			(*Robot 21*)
			IF (Human_Reqs_TraccTCP_R21)
					AND ((NOT Start_All_MTRobots AND NOT Start_All_BTRobots
					AND NOT Start_All_TCRobots AND NOT Start_All_TDRobots)
					OR (MAIN.R21.Task_ID_Ack=Tracc_TCP))
				THEN
					(*Start Robot*)
					Start_TraccTCP_21:= TRUE;
					(*Allow Robot to Proceed*)
					TraccRobot_21_Proceed:= TRUE;
			ELSE
					Start_TraccTCP_21:= FALSE;
					TraccRobot_21_Proceed:= FALSE;
			END_IF;	
			
			(*Robot 22*)
			IF (Human_Reqs_TraccTCP_R22)
					AND ((NOT Start_All_MTRobots AND NOT Start_All_BTRobots
					AND NOT Start_All_TCRobots AND NOT Start_All_TDRobots)
					OR (MAIN.R22.Task_ID_Ack=Tracc_TCP))
				THEN
					(*Start Robot*)
					Start_TraccTCP_22:= TRUE;
					(*Allow Robot to Proceed*)
					TraccRobot_22_Proceed:= TRUE;
			ELSE
					Start_TraccTCP_22:= FALSE;
					TraccRobot_22_Proceed:= FALSE;
			END_IF;	
			
			(*Robot 23*)
			IF (Human_Reqs_TraccTCP_R23)
					AND ((NOT Start_All_MTRobots AND NOT Start_All_BTRobots
					AND NOT Start_All_TCRobots AND NOT Start_All_TDRobots)
					OR (MAIN.R23.Task_ID_Ack=Tracc_TCP))
				THEN
					(*Start Robot*)
					Start_TraccTCP_23:= TRUE;
					(*Allow Robot to Proceed*)
					TraccRobot_23_Proceed:= TRUE;
			ELSE
					Start_TraccTCP_23:= FALSE;
					TraccRobot_23_Proceed:= FALSE;
			END_IF;	
			
			(*Robot 24*)
			IF (Human_Reqs_TraccTCP_R24)
					AND ((NOT Start_All_MTRobots AND NOT Start_All_BTRobots
					AND NOT Start_All_TCRobots AND NOT Start_All_TDRobots)
					OR (MAIN.R24.Task_ID_Ack=Tracc_TCP))
				THEN
					(*Start Robot*)
					Start_TraccTCP_24:= TRUE;
					(*Allow Robot to Proceed*)
					TraccRobot_24_Proceed:= TRUE;
			ELSE
					Start_TraccTCP_24:= FALSE;
					TraccRobot_24_Proceed:= FALSE;
			END_IF;	
			
			(*Robot 25*)
			IF (Human_Reqs_TraccTCP_R25)
					AND ((NOT Start_All_MTRobots AND NOT Start_All_BTRobots
					AND NOT Start_All_TCRobots AND NOT Start_All_TDRobots)
					OR (MAIN.R25.Task_ID_Ack=Tracc_TCP))
				THEN
					(*Start Robot*)
					Start_TraccTCP_25:= TRUE;
					(*Allow Robot to Proceed*)
					TraccRobot_25_Proceed:= TRUE;
			ELSE
					Start_TraccTCP_25:= FALSE;
					TraccRobot_25_Proceed:= FALSE;
			END_IF;	
			
			(*Robot 26*)
			IF (Human_Reqs_TraccTCP_R26)
					AND ((NOT Start_All_MTRobots AND NOT Start_All_BTRobots
					AND NOT Start_All_TCRobots AND NOT Start_All_TDRobots)
					OR (MAIN.R26.Task_ID_Ack=Tracc_TCP))
				THEN
					(*Start Robot*)
					Start_TraccTCP_26:= TRUE;
					(*Allow Robot to Proceed*)
					TraccRobot_26_Proceed:= TRUE;
			ELSE
					Start_TraccTCP_26:= FALSE;
					TraccRobot_26_Proceed:= FALSE;
			END_IF;	
			
			(*Robot 27*)
			IF (Human_Reqs_TraccTCP_R27)
					AND ((NOT Start_All_MTRobots AND NOT Start_All_BTRobots
					AND NOT Start_All_TCRobots AND NOT Start_All_TDRobots)
					OR (MAIN.R27.Task_ID_Ack=Tracc_TCP))
				THEN
					(*Start Robot*)
					Start_TraccTCP_27:= TRUE;
					(*Allow Robot to Proceed*)
					TraccRobot_27_Proceed:= TRUE;
			ELSE
					Start_TraccTCP_27:= FALSE;
					TraccRobot_27_Proceed:= FALSE;
			END_IF;	
			
			(*Robot 28*)
			IF (Human_Reqs_TraccTCP_R28)
					AND ((NOT Start_All_MTRobots AND NOT Start_All_BTRobots
					AND NOT Start_All_TCRobots AND NOT Start_All_TDRobots)
					OR (MAIN.R28.Task_ID_Ack=Tracc_TCP))
				THEN
					(*Start Robot*)
					Start_TraccTCP_28:= TRUE;
					(*Allow Robot to Proceed*)
					TraccRobot_28_Proceed:= TRUE;
			ELSE
					Start_TraccTCP_28:= FALSE;
					TraccRobot_28_Proceed:= FALSE;
			END_IF;	
			
			(*Robot 29*)
			IF (Human_Reqs_TraccTCP_R29)
					AND ((NOT Start_All_MTRobots AND NOT Start_All_BTRobots
					AND NOT Start_All_TCRobots AND NOT Start_All_TDRobots)
					OR (MAIN.R29.Task_ID_Ack=Tracc_TCP))
				THEN
					(*Start Robot*)
					Start_TraccTCP_29:= TRUE;
					(*Allow Robot to Proceed*)
					TraccRobot_29_Proceed:= TRUE;
			ELSE
					Start_TraccTCP_29:= FALSE;
					TraccRobot_29_Proceed:= FALSE;
			END_IF;
			
			(*Robot 30*)
			IF (Human_Reqs_TraccTCP_R30)
					AND ((NOT Start_All_MTRobots AND NOT Start_All_BTRobots
					AND NOT Start_All_TCRobots AND NOT Start_All_TDRobots)
					OR (MAIN.R30.Task_ID_Ack=Tracc_TCP))
				THEN
					(*Start Robot*)
					Start_TraccTCP_30:= TRUE;
					(*Allow Robot to Proceed*)
					TraccRobot_30_Proceed:= TRUE;
			ELSE
					Start_TraccTCP_30:= FALSE;
					TraccRobot_30_Proceed:= FALSE;
			END_IF;	
				

			
			
			
	ELSE
		Start_All_MTRobots:= FALSE;
		Start_All_BTRobots:= FALSE;
		Start_All_TCRobots:= FALSE;
		Start_All_TDRobots:= FALSE;
		Start_TDRobot_1:= FALSE;
		Start_TDRobot_2:= FALSE;
		Start_TDRobot_3:= FALSE;
		Start_TDRobot_4:= FALSE;
		Start_TDRobot_5:= FALSE;
		Start_TDRobot_6:= FALSE;
		Start_TDRobot_7:= FALSE;
		Start_TDRobot_8:= FALSE;
		Start_TDRobot_9:= FALSE;
		Start_TDRobot_10:= FALSE;
		Start_TDRobot_11:= FALSE;
		Start_TDRobot_12:= FALSE;
		Start_TDRobot_13:= FALSE;
		Start_TDRobot_14:= FALSE;
		Start_TDRobot_15:= FALSE;
		Start_TDRobot_16:= FALSE;
		Start_TDRobot_17:= FALSE;
		Start_TDRobot_18:= FALSE;
		Start_TDRobot_19:= FALSE;
		Start_TDRobot_20:= FALSE;
		Start_TDRobot_21:= FALSE;
		Start_TDRobot_22:= FALSE;
		Start_TDRobot_23:= FALSE;
		Start_TDRobot_24:= FALSE;
		Start_TDRobot_25:= FALSE;
		Start_TDRobot_26:= FALSE;
		Start_TDRobot_27:= FALSE;
		Start_TDRobot_28:= FALSE;
		Start_TDRobot_29:= FALSE;
		Start_TDRobot_30:= FALSE;
		Start_All_TraccTCP:= FALSE;
		Start_TraccTCP_1:= FALSE;
		Start_TraccTCP_2:= FALSE;
		Start_TraccTCP_3:= FALSE;
		Start_TraccTCP_4:= FALSE;
		Start_TraccTCP_5:= FALSE;
		Start_TraccTCP_6:= FALSE;
		Start_TraccTCP_7:= FALSE;
		Start_TraccTCP_8:= FALSE;
		Start_TraccTCP_9:= FALSE;
		Start_TraccTCP_10:= FALSE;
		Start_TraccTCP_11:= FALSE;
		Start_TraccTCP_12:= FALSE;
		Start_TraccTCP_13:= FALSE;
		Start_TraccTCP_14:= FALSE;
		Start_TraccTCP_15:= FALSE;
		Start_TraccTCP_16:= FALSE;
		Start_TraccTCP_17:= FALSE;
		Start_TraccTCP_18:= FALSE;
		Start_TraccTCP_19:= FALSE;
		Start_TraccTCP_20:= FALSE;
		Start_TraccTCP_21:= FALSE;
		Start_TraccTCP_22:= FALSE;
		Start_TraccTCP_23:= FALSE;
		Start_TraccTCP_24:= FALSE;
		Start_TraccTCP_25:= FALSE;
		Start_TraccTCP_26:= FALSE;
		Start_TraccTCP_27:= FALSE;
		Start_TraccTCP_28:= FALSE;
		Start_TraccTCP_29:= FALSE;
		Start_TraccTCP_30:= FALSE;
	END_IF;

(*---------------------------------------------------------------Completes----------------------------------------------------*)
	(*All Robots Complete Master Test*)
	IF Start_All_MTRobots AND All_Robots_Complete
		THEN
		Master_Tests_Complete:= TRUE;
		Human_Reqs_MasterTest:= FALSE;
		A_Robot_Reqs_MasterTest:= FALSE;
	END_IF;
	(*All Robots Complete Brake Test*)
	IF Start_All_BTRobots AND All_Robots_Complete
		THEN
		Brake_Tests_Complete:= TRUE;
		Human_Reqs_BrakeTest:= FALSE;
		A_Robot_Reqs_BrakeTest:= FALSE;
		All_RobotsReq_BrakeTest:= FALSE;
	END_IF;
	(*All Robots Complete Tip Change*)
	IF Start_All_TCRobots AND All_Robots_SteppersRST AND All_Robots_Complete
		THEN
		Tip_Change_Complete:= TRUE;
		Human_Reqs_TipChange:= FALSE;
	         Robot_Reqs_TipChange := FALSE;
	END_IF;

	(*All Robots Complete Tip Dress*)
	IF Start_All_TDRobots AND All_Robots_Complete
		THEN
		Tip_Dress_CompleteAll:= TRUE;
		TipChange_Reqs_TipDress:= FALSE;
		Robot_Reqs_TipDress:= FALSE;
	END_IF;

	(*Robot1 Complete Tip Dress*)
	IF Tip_Dress_Complete1
		THEN
		Human_Reqs_TipDressR1:= FALSE;
		Robot1_Reqs_TipDress:= FALSE;
	END_IF;

	(*Robot2 Complete Tip Dress*)
	IF Tip_Dress_Complete2
		THEN
		Human_Reqs_TipDressR2:= FALSE;
		Robot2_Reqs_TipDress:= FALSE;
	END_IF;

	(*Robot3 Complete Tip Dress*)
	IF Tip_Dress_Complete3
		THEN
		Human_Reqs_TipDressR3:= FALSE;
		Robot3_Reqs_TipDress:= FALSE;
	END_IF;

	(*Robot4 Complete Tip Dress*)
	IF Tip_Dress_Complete4
		THEN
		Human_Reqs_TipDressR4:= FALSE;
		Robot4_Reqs_TipDress:= FALSE;
	END_IF;

	(*Robot5 Complete Tip Dress*)
	IF Tip_Dress_Complete5
		THEN
		Human_Reqs_TipDressR5:= FALSE;
		Robot5_Reqs_TipDress:= FALSE;
	END_IF;

	(*Robot6 Complete Tip Dress*)
	IF Tip_Dress_Complete6
		THEN
		Human_Reqs_TipDressR6:= FALSE;
		Robot6_Reqs_TipDress:= FALSE;
	END_IF;

	(*Robot7 Complete Tip Dress*)
	IF Tip_Dress_Complete7
		THEN
		Human_Reqs_TipDressR7:= FALSE;
		Robot7_Reqs_TipDress:= FALSE;
	END_IF;

	(*Robot8 Complete Tip Dress*)
	IF Tip_Dress_Complete8
		THEN
		Human_Reqs_TipDressR8:= FALSE;
		Robot8_Reqs_TipDress:= FALSE;
	END_IF;

	(*Robot9 Complete Tip Dress*)
	IF Tip_Dress_Complete9
		THEN
		Human_Reqs_TipDressR9:= FALSE;
		Robot9_Reqs_TipDress:= FALSE;
	END_IF;

	(*Robot10 Complete Tip Dress*)
	IF Tip_Dress_Complete10
		THEN
		Human_Reqs_TipDressR10:= FALSE;
		Robot10_Reqs_TipDress:= FALSE;
	END_IF;

	(*Robot11 Complete Tip Dress*)
	IF Tip_Dress_Complete11
		THEN
		Human_Reqs_TipDressR11:= FALSE;
		Robot11_Reqs_TipDress:= FALSE;
	END_IF;

	(*Robot12 Complete Tip Dress*)
	IF Tip_Dress_Complete12
		THEN
		Human_Reqs_TipDressR12:= FALSE;
		Robot12_Reqs_TipDress:= FALSE;
	END_IF;

	(*Robot13 Complete Tip Dress*)
	IF Tip_Dress_Complete13
		THEN
		Human_Reqs_TipDressR13:= FALSE;
		Robot13_Reqs_TipDress:= FALSE;
	END_IF;

	(*Robot14 Complete Tip Dress*)
	IF Tip_Dress_Complete14
		THEN
		Human_Reqs_TipDressR14:= FALSE;
		Robot14_Reqs_TipDress:= FALSE;
	END_IF;

	(*Robot15 Complete Tip Dress*)
	IF Tip_Dress_Complete15
		THEN
		Human_Reqs_TipDressR15:= FALSE;
		Robot15_Reqs_TipDress:= FALSE;
	END_IF;

	(*Robot16 Complete Tip Dress*)
	IF Tip_Dress_Complete16
		THEN
		Human_Reqs_TipDressR16:= FALSE;
		Robot16_Reqs_TipDress:= FALSE;
	END_IF;

	(*Robot17 Complete Tip Dress*)
	IF Tip_Dress_Complete17
		THEN
		Human_Reqs_TipDressR17:= FALSE;
		Robot17_Reqs_TipDress:= FALSE;
	END_IF;

	(*Robot18 Complete Tip Dress*)
	IF Tip_Dress_Complete18
		THEN
		Human_Reqs_TipDressR18:= FALSE;
		Robot18_Reqs_TipDress:= FALSE;
	END_IF;

	(*Robot19 Complete Tip Dress*)
	IF Tip_Dress_Complete19
		THEN
		Human_Reqs_TipDressR19:= FALSE;
		Robot19_Reqs_TipDress:= FALSE;
	END_IF;

	(*Robot20 Complete Tip Dress*)
	IF Tip_Dress_Complete20
		THEN
		Human_Reqs_TipDressR20:= FALSE;
		Robot20_Reqs_TipDress:= FALSE;
	END_IF;

	(*Robot21 Complete Tip Dress*)
	IF Tip_Dress_Complete21
		THEN
		Human_Reqs_TipDressR21:= FALSE;
		Robot21_Reqs_TipDress:= FALSE;
	END_IF;

	(*Robot22 Complete Tip Dress*)
	IF Tip_Dress_Complete22
		THEN
		Human_Reqs_TipDressR22:= FALSE;
		Robot22_Reqs_TipDress:= FALSE;
	END_IF;

	(*Robot23 Complete Tip Dress*)
	IF Tip_Dress_Complete23
		THEN
		Human_Reqs_TipDressR23:= FALSE;
		Robot23_Reqs_TipDress:= FALSE;
	END_IF;

	(*Robot24 Complete Tip Dress*)
	IF Tip_Dress_Complete24
		THEN
		Human_Reqs_TipDressR24:= FALSE;
		Robot24_Reqs_TipDress:= FALSE;
	END_IF;

	(*Robot25 Complete Tip Dress*)
	IF Tip_Dress_Complete25
		THEN
		Human_Reqs_TipDressR25:= FALSE;
		Robot25_Reqs_TipDress:= FALSE;
	END_IF;

	(*Robot26 Complete Tip Dress*)
	IF Tip_Dress_Complete26
		THEN
		Human_Reqs_TipDressR26:= FALSE;
		Robot26_Reqs_TipDress:= FALSE;
	END_IF;

	(*Robot27 Complete Tip Dress*)
	IF Tip_Dress_Complete27
		THEN
		Human_Reqs_TipDressR27:= FALSE;
		Robot27_Reqs_TipDress:= FALSE;
	END_IF;

	(*Robot28 Complete Tip Dress*)
	IF Tip_Dress_Complete28
		THEN
		Human_Reqs_TipDressR28:= FALSE;
		Robot28_Reqs_TipDress:= FALSE;
	END_IF;

	(*Robot29 Complete Tip Dress*)
	IF Tip_Dress_Complete29
		THEN
		Human_Reqs_TipDressR29:= FALSE;
		Robot29_Reqs_TipDress:= FALSE;
	END_IF;

	(*Robot30 Complete Tip Dress*)
	IF Tip_Dress_Complete30
		THEN
		Human_Reqs_TipDressR30:= FALSE;
		Robot30_Reqs_TipDress:= FALSE;
	END_IF;

	(*Robot 1 Complete TraccTCP*)
	IF TraccTCP_Complete1
		THEN
		Human_Reqs_TraccTCP_R1:= FALSE;
		Robot1_Reqs_TraccTCP:= FALSE;
	END_IF;

	(*Robot 2 Complete TraccTCP*)
	IF TraccTCP_Complete2
		THEN
		Human_Reqs_TraccTCP_R2:= FALSE;
		Robot2_Reqs_TraccTCP:= FALSE;
	END_IF;

	(*Robot 3 Complete TraccTCP*)
	IF TraccTCP_Complete3
		THEN
		Human_Reqs_TraccTCP_R3:= FALSE;
		Robot3_Reqs_TraccTCP:= FALSE;
	END_IF;

	(*Robot 4 Complete TraccTCP*)
	IF TraccTCP_Complete4
		THEN
		Human_Reqs_TraccTCP_R4:= FALSE;
		Robot4_Reqs_TraccTCP:= FALSE;
	END_IF;	

	(*Robot 5 Complete TraccTCP*)
	IF TraccTCP_Complete5
		THEN
		Human_Reqs_TraccTCP_R5:= FALSE;
		Robot5_Reqs_TraccTCP:= FALSE;
	END_IF;

	(*Robot 6 Complete TraccTCP*)
	IF TraccTCP_Complete6
		THEN
		Human_Reqs_TraccTCP_R6:= FALSE;
		Robot6_Reqs_TraccTCP:= FALSE;
	END_IF;

	(*Robot 7 Complete TraccTCP*)
	IF TraccTCP_Complete7
		THEN
		Human_Reqs_TraccTCP_R7:= FALSE;
		Robot7_Reqs_TraccTCP:= FALSE;
	END_IF;
	
	(*Robot 8 Complete TraccTCP*)
	IF TraccTCP_Complete8
		THEN
		Human_Reqs_TraccTCP_R8:= FALSE;
		Robot8_Reqs_TraccTCP:= FALSE;
	END_IF;
	
	(*Robot 9 Complete TraccTCP*)
	IF TraccTCP_Complete9
		THEN
		Human_Reqs_TraccTCP_R9:= FALSE;
		Robot9_Reqs_TraccTCP:= FALSE;
	END_IF;
	
	(*Robot 10 Complete TraccTCP*)
	IF TraccTCP_Complete10
		THEN
		Human_Reqs_TraccTCP_R10:= FALSE;
		Robot10_Reqs_TraccTCP:= FALSE;
	END_IF;

	(*Robot 11 Complete TraccTCP*)
	IF TraccTCP_Complete11
		THEN
		Human_Reqs_TraccTCP_R11:= FALSE;
		Robot11_Reqs_TraccTCP:= FALSE;
	END_IF;
	
	(*Robot 12 Complete TraccTCP*)
	IF TraccTCP_Complete12
		THEN
		Human_Reqs_TraccTCP_R12:= FALSE;
		Robot12_Reqs_TraccTCP:= FALSE;
	END_IF;
	
	(*Robot 13 Complete TraccTCP*)
	IF TraccTCP_Complete13
		THEN
		Human_Reqs_TraccTCP_R13:= FALSE;
		Robot13_Reqs_TraccTCP:= FALSE;
	END_IF;
	
	(*Robot 14 Complete TraccTCP*)
	IF TraccTCP_Complete14
		THEN
		Human_Reqs_TraccTCP_R14:= FALSE;
		Robot14_Reqs_TraccTCP:= FALSE;
	END_IF;
	
	(*Robot 15 Complete TraccTCP*)
	IF TraccTCP_Complete15
		THEN
		Human_Reqs_TraccTCP_R15:= FALSE;
		Robot15_Reqs_TraccTCP:= FALSE;
	END_IF;
	
	(*Robot 16 Complete TraccTCP*)
	IF TraccTCP_Complete16
		THEN
		Human_Reqs_TraccTCP_R16:= FALSE;
		Robot16_Reqs_TraccTCP:= FALSE;
	END_IF;
	
	(*Robot 17 Complete TraccTCP*)
	IF TraccTCP_Complete17
		THEN
		Human_Reqs_TraccTCP_R17:= FALSE;
		Robot17_Reqs_TraccTCP:= FALSE;
	END_IF;
	
	(*Robot 18 Complete TraccTCP*)
	IF TraccTCP_Complete18
		THEN
		Human_Reqs_TraccTCP_R18:= FALSE;
		Robot18_Reqs_TraccTCP:= FALSE;
	END_IF;
	
	(*Robot 19 Complete TraccTCP*)
	IF TraccTCP_Complete19
		THEN
		Human_Reqs_TraccTCP_R19:= FALSE;
		Robot19_Reqs_TraccTCP:= FALSE;
	END_IF;
	
	(*Robot 20 Complete TraccTCP*)
	IF TraccTCP_Complete20
		THEN
		Human_Reqs_TraccTCP_R20:= FALSE;
		Robot20_Reqs_TraccTCP:= FALSE;
	END_IF;

	(*Robot 21 Complete TraccTCP*)
	IF TraccTCP_Complete21
		THEN
		Human_Reqs_TraccTCP_R21:= FALSE;
		Robot21_Reqs_TraccTCP:= FALSE;
	END_IF;
	
	(*Robot 22 Complete TraccTCP*)
	IF TraccTCP_Complete22
		THEN
		Human_Reqs_TraccTCP_R22:= FALSE;
		Robot22_Reqs_TraccTCP:= FALSE;
	END_IF;
	
	(*Robot 23 Complete TraccTCP*)
	IF TraccTCP_Complete23
		THEN
		Human_Reqs_TraccTCP_R23:= FALSE;
		Robot23_Reqs_TraccTCP:= FALSE;
	END_IF;
	
	(*Robot 24 Complete TraccTCP*)
	IF TraccTCP_Complete24
		THEN
		Human_Reqs_TraccTCP_R24:= FALSE;
		Robot24_Reqs_TraccTCP:= FALSE;
	END_IF;
	
	(*Robot 25 Complete TraccTCP*)
	IF TraccTCP_Complete25
		THEN
		Human_Reqs_TraccTCP_R25:= FALSE;
		Robot25_Reqs_TraccTCP:= FALSE;
	END_IF;
	
	(*Robot 26 Complete TraccTCP*)
	IF TraccTCP_Complete26
		THEN
		Human_Reqs_TraccTCP_R26:= FALSE;
		Robot26_Reqs_TraccTCP:= FALSE;
	END_IF;
	
	(*Robot 27 Complete TraccTCP*)
	IF TraccTCP_Complete27
		THEN
		Human_Reqs_TraccTCP_R27:= FALSE;
		Robot27_Reqs_TraccTCP:= FALSE;
	END_IF;
	
	(*Robot 28 Complete TraccTCP*)
	IF TraccTCP_Complete28
		THEN
		Human_Reqs_TraccTCP_R28:= FALSE;
		Robot28_Reqs_TraccTCP:= FALSE;
	END_IF;
	
	(*Robot 29 Complete TraccTCP*)
	IF TraccTCP_Complete29
		THEN
		Human_Reqs_TraccTCP_R29:= FALSE;
		Robot29_Reqs_TraccTCP:= FALSE;
	END_IF;
	
	(*Robot 30 Complete TraccTCP*)
	IF TraccTCP_Complete30
		THEN
		Human_Reqs_TraccTCP_R30:= FALSE;
		Robot30_Reqs_TraccTCP:= FALSE;
	END_IF;
	
	
	
(*!!!!!!!!!!!!!!!!!!!!!!!!!!!!!!!!!!!!!!!!!!!!!!!!!!!!!!!!!!!!!!!!!!!!!!!!!!!!!!!!!!!!!!!!!!!!!!!!! Cycle Complete !!!!!!!!!!!!!!!!!!!!!!!!!!!!!!!!!!!!!!!!!!!!!!!!!!!!!!!!!!!!!!!!!!!!!!!!!!!!!!!!!!!!!!!!!!*)
	(*Set Cycle Complete*)
	IF Auto_Run AND (Master_Tests_Complete OR Brake_Tests_Complete OR Tip_Change_Complete OR Tip_Dress_CompleteAll OR TraccTCP_CompleteAll)
		THEN Cycle_Complete:= TRUE;
	END_IF;
	(*Reset All Completes*)
	IF Cycle_Complete AND All_Robots_Clear
		THEN
					Reset_All_Completes:= TRUE;
	END_IF;
	(*Perform Actual Reset*)
		IF Reset_All_Completes
			THEN
				Cycle_Complete:= FALSE;
				Human_Reqs_MasterTest := FALSE;
				A_Robot_Reqs_MasterTest :=FALSE;
				Master_Tests_Complete:= FALSE;
				Human_Reqs_BrakeTest := FALSE;
				A_Robot_Reqs_BrakeTest := FALSE;
				All_RobotsReq_BrakeTest := FALSE;
				Brake_Tests_Complete:= FALSE;
				Tip_Change_Complete:= FALSE;
				Tip_Dress_CompleteAll:= FALSE;
				TraccTCP_CompleteAll:= FALSE;
				Reset_All_Completes:= FALSE;
		END_IF;

(*$$$$$$$$$$$$$$$$$$$$$$$$$$$$$$$$$$$ Production Counter $$$$$$$$$$$$$$$$$$$$$$$$$$$$$$$$$$$$$$$$$$*)
	(*Increment Tip Change Counter*)
	Prod_Inc.CLK:= Tip_Change_Complete;
	Prod_Inc();
	IF Prod_Inc.Q
		THEN
		Production_Count:= Production_Count+1;
	END_IF;
	IF Discrete_In.ResetProd
		THEN
		Production_Count:= 0;
	END_IF;
	Prod_Count_Out:= Production_Count;
(*~~~~~~~~~~~~~~~~~~~~~~~~~~~~~~~~ Cycle Time Counters ~~~~~~~~~~~~~~~~~~~~~~~~~*)
	(*Move Previous To Register*)
	Cycle_Time_Pulse.CLK:= Tip_Change_Complete;
	Cycle_Time_Pulse();
	IF Cycle_Time_Pulse.Q
		THEN
		PrevCycle_Time_Out:= Cycle_Time_Out;
	END_IF;
	(*Monitor Current Cycle Time*)
		Cycle_Time.PT:= T#9999S;
		Cycle_Time.IN:= Auto_Run AND NOT Cycle_Complete;
		Cycle_Time();
		Cycle_Time_Out:= Cycle_Time.ET;

(*^^^^^^^^^^^^^^^^^^^^^^^^^^^^^^^^^^^^^^ General Visualization ^^^^^^^^^^^^^^^^^^^^^^^^^^^^^^^^^^^^*)

(*#################################### Register Robots to Tool ##################################*)
(*+++++++++++THIS AREA IS CUSTOM PER INSTALLATION AND WILL HAVE TO BE MODIFIED PER +++++++++++++*)
(*+++++++++++THIS AREA IS CUSTOM PER INSTALLATION AND WILL HAVE TO BE MODIFIED PER +++++++++++++*)

	(*Data From All Robot(s)*)

	All_Robots_Clear:= MAIN.R1.Clear_Of_EquipInterf8 AND MAIN.R1.Task_ID_Ack<350 AND
					(MAIN.R2.Clear_Of_EquipInterf8 AND MAIN.R2.Task_ID_Ack<350 OR GTAC_CONFIG.Option_Robot_Count<2) AND
					(MAIN.R3.Clear_Of_EquipInterf8 AND MAIN.R3.Task_ID_Ack<350 OR GTAC_CONFIG.Option_Robot_Count<3) AND
					(MAIN.R4.Clear_Of_EquipInterf8 AND MAIN.R4.Task_ID_Ack<350 OR GTAC_CONFIG.Option_Robot_Count<4) AND
					(MAIN.R5.Clear_Of_EquipInterf8 AND MAIN.R5.Task_ID_Ack<350 OR GTAC_CONFIG.Option_Robot_Count<5) AND
					(MAIN.R6.Clear_Of_EquipInterf8 AND MAIN.R6.Task_ID_Ack<350 OR GTAC_CONFIG.Option_Robot_Count<6) AND
					(MAIN.R7.Clear_Of_EquipInterf8 AND MAIN.R7.Task_ID_Ack<350 OR GTAC_CONFIG.Option_Robot_Count<7) AND
					(MAIN.R8.Clear_Of_EquipInterf8 AND MAIN.R8.Task_ID_Ack<350 OR GTAC_CONFIG.Option_Robot_Count<8) AND
					(MAIN.R9.Clear_Of_EquipInterf8 AND MAIN.R9.Task_ID_Ack<350 OR GTAC_CONFIG.Option_Robot_Count<9) AND
					(MAIN.R10.Clear_Of_EquipInterf8 AND MAIN.R10.Task_ID_Ack<350 OR GTAC_CONFIG.Option_Robot_Count<10) AND
					(MAIN.R11.Clear_Of_EquipInterf8 AND MAIN.R11.Task_ID_Ack<350 OR GTAC_CONFIG.Option_Robot_Count<11) AND
					(MAIN.R12.Clear_Of_EquipInterf8 AND MAIN.R12.Task_ID_Ack<350 OR GTAC_CONFIG.Option_Robot_Count<12) AND
					(MAIN.R13.Clear_Of_EquipInterf8 AND MAIN.R13.Task_ID_Ack<350 OR GTAC_CONFIG.Option_Robot_Count<13) AND
					(MAIN.R14.Clear_Of_EquipInterf8 AND MAIN.R14.Task_ID_Ack<350 OR GTAC_CONFIG.Option_Robot_Count<14) AND
					(MAIN.R15.Clear_Of_EquipInterf8 AND MAIN.R15.Task_ID_Ack<350 OR GTAC_CONFIG.Option_Robot_Count<15) AND
					(MAIN.R16.Clear_Of_EquipInterf8 AND MAIN.R16.Task_ID_Ack<350 OR GTAC_CONFIG.Option_Robot_Count<16) AND
					(MAIN.R17.Clear_Of_EquipInterf8 AND MAIN.R17.Task_ID_Ack<350 OR GTAC_CONFIG.Option_Robot_Count<17) AND
					(MAIN.R18.Clear_Of_EquipInterf8 AND MAIN.R18.Task_ID_Ack<350 OR GTAC_CONFIG.Option_Robot_Count<18) AND
					(MAIN.R19.Clear_Of_EquipInterf8 AND MAIN.R19.Task_ID_Ack<350 OR GTAC_CONFIG.Option_Robot_Count<19) AND
					(MAIN.R20.Clear_Of_EquipInterf8 AND MAIN.R20.Task_ID_Ack<350 OR GTAC_CONFIG.Option_Robot_Count<20) AND
					(MAIN.R21.Clear_Of_EquipInterf8 AND MAIN.R21.Task_ID_Ack<350 OR GTAC_CONFIG.Option_Robot_Count<21) AND
					(MAIN.R22.Clear_Of_EquipInterf8 AND MAIN.R22.Task_ID_Ack<350 OR GTAC_CONFIG.Option_Robot_Count<22) AND
					(MAIN.R23.Clear_Of_EquipInterf8 AND MAIN.R23.Task_ID_Ack<350 OR GTAC_CONFIG.Option_Robot_Count<23) AND
					(MAIN.R24.Clear_Of_EquipInterf8 AND MAIN.R24.Task_ID_Ack<350 OR GTAC_CONFIG.Option_Robot_Count<24) AND
					(MAIN.R25.Clear_Of_EquipInterf8 AND MAIN.R25.Task_ID_Ack<350 OR GTAC_CONFIG.Option_Robot_Count<25) AND
					(MAIN.R26.Clear_Of_EquipInterf8 AND MAIN.R26.Task_ID_Ack<350 OR GTAC_CONFIG.Option_Robot_Count<26) AND
					(MAIN.R27.Clear_Of_EquipInterf8 AND MAIN.R27.Task_ID_Ack<350 OR GTAC_CONFIG.Option_Robot_Count<27) AND
					(MAIN.R28.Clear_Of_EquipInterf8 AND MAIN.R28.Task_ID_Ack<350 OR GTAC_CONFIG.Option_Robot_Count<28) AND
					(MAIN.R29.Clear_Of_EquipInterf8 AND MAIN.R29.Task_ID_Ack<350 OR GTAC_CONFIG.Option_Robot_Count<29) AND
					(MAIN.R30.Clear_Of_EquipInterf8 AND MAIN.R30.Task_ID_Ack<350 OR GTAC_CONFIG.Option_Robot_Count<30);

	All_Robots_WorkingOK:=  (Start_All_MTRobots AND MAIN.R1.Task_ID_Ack=Master_Test AND MAIN.R1.Operating AND
											(MAIN.R2.Task_ID_Ack=Master_Test AND MAIN.R2.Operating OR GTAC_CONFIG.Option_Robot_Count<2) AND
											(MAIN.R3.Task_ID_Ack=Master_Test AND MAIN.R3.Operating OR GTAC_CONFIG.Option_Robot_Count<3) AND
											(MAIN.R4.Task_ID_Ack=Master_Test AND MAIN.R4.Operating OR GTAC_CONFIG.Option_Robot_Count<4) AND
											(MAIN.R5.Task_ID_Ack=Master_Test AND MAIN.R5.Operating OR GTAC_CONFIG.Option_Robot_Count<5) AND
											(MAIN.R6.Task_ID_Ack=Master_Test AND MAIN.R6.Operating OR GTAC_CONFIG.Option_Robot_Count<6) AND
											(MAIN.R7.Task_ID_Ack=Master_Test AND MAIN.R7.Operating OR GTAC_CONFIG.Option_Robot_Count<7) AND
											(MAIN.R8.Task_ID_Ack= Master_Test AND MAIN.R8.Operating OR GTAC_CONFIG.Option_Robot_Count<8) AND
											(MAIN.R9.Task_ID_Ack=Master_Test AND MAIN.R9.Operating OR GTAC_CONFIG.Option_Robot_Count<9) AND
											(MAIN.R10.Task_ID_Ack= Master_Test AND MAIN.R10.Operating OR GTAC_CONFIG.Option_Robot_Count<10) AND
											(MAIN.R11.Task_ID_Ack=Master_Test AND MAIN.R11.Operating OR GTAC_CONFIG.Option_Robot_Count<11) AND
											(MAIN.R12.Task_ID_Ack=Master_Test AND MAIN.R12.Operating OR GTAC_CONFIG.Option_Robot_Count<12) AND
											(MAIN.R13.Task_ID_Ack=Master_Test AND MAIN.R13.Operating OR GTAC_CONFIG.Option_Robot_Count<13) AND
											(MAIN.R14.Task_ID_Ack=Master_Test AND MAIN.R14.Operating OR GTAC_CONFIG.Option_Robot_Count<14) AND
											(MAIN.R15.Task_ID_Ack=Master_Test AND MAIN.R15.Operating OR GTAC_CONFIG.Option_Robot_Count<15) AND
											(MAIN.R16.Task_ID_Ack=Master_Test AND MAIN.R16.Operating OR GTAC_CONFIG.Option_Robot_Count<16) AND
											(MAIN.R17.Task_ID_Ack=Master_Test AND MAIN.R17.Operating OR GTAC_CONFIG.Option_Robot_Count<17) AND
											(MAIN.R18.Task_ID_Ack= Master_Test AND MAIN.R18.Operating OR GTAC_CONFIG.Option_Robot_Count<18) AND
											(MAIN.R19.Task_ID_Ack=Master_Test AND MAIN.R19.Operating OR GTAC_CONFIG.Option_Robot_Count<19) AND
											(MAIN.R20.Task_ID_Ack=Master_Test AND MAIN.R20.Operating OR GTAC_CONFIG.Option_Robot_Count<20) AND
											(MAIN.R21.Task_ID_Ack=Master_Test AND MAIN.R21.Operating OR GTAC_CONFIG.Option_Robot_Count<21) AND
											(MAIN.R22.Task_ID_Ack=Master_Test AND MAIN.R22.Operating OR GTAC_CONFIG.Option_Robot_Count<22) AND
											(MAIN.R23.Task_ID_Ack=Master_Test AND MAIN.R23.Operating OR GTAC_CONFIG.Option_Robot_Count<23) AND
											(MAIN.R24.Task_ID_Ack=Master_Test AND MAIN.R24.Operating OR GTAC_CONFIG.Option_Robot_Count<24) AND
											(MAIN.R25.Task_ID_Ack=Master_Test AND MAIN.R25.Operating OR GTAC_CONFIG.Option_Robot_Count<25) AND
											(MAIN.R26.Task_ID_Ack=Master_Test AND MAIN.R26.Operating OR GTAC_CONFIG.Option_Robot_Count<26) AND
											(MAIN.R27.Task_ID_Ack=Master_Test AND MAIN.R27.Operating OR GTAC_CONFIG.Option_Robot_Count<27) AND
											(MAIN.R28.Task_ID_Ack=Master_Test AND MAIN.R28.Operating OR GTAC_CONFIG.Option_Robot_Count<28) AND
											(MAIN.R29.Task_ID_Ack=Master_Test AND MAIN.R29.Operating OR GTAC_CONFIG.Option_Robot_Count<29) AND
											(MAIN.R30.Task_ID_Ack=Master_Test AND MAIN.R30.Operating OR GTAC_CONFIG.Option_Robot_Count<30))
											OR
							(Start_All_BTRobots AND MAIN.R1.Task_ID_Ack=Brake_Test AND MAIN.R1.Operating AND
											(MAIN.R2.Task_ID_Ack=Brake_Test AND MAIN.R2.Operating OR GTAC_CONFIG.Option_Robot_Count<2) AND
											(MAIN.R3.Task_ID_Ack=Brake_Test AND MAIN.R3.Operating OR GTAC_CONFIG.Option_Robot_Count<3) AND
											(MAIN.R4.Task_ID_Ack=Brake_Test AND MAIN.R4.Operating OR GTAC_CONFIG.Option_Robot_Count<4) AND
											(MAIN.R5.Task_ID_Ack=Brake_Test AND MAIN.R5.Operating OR GTAC_CONFIG.Option_Robot_Count<5) AND
											(MAIN.R6.Task_ID_Ack=Brake_Test AND MAIN.R6.Operating OR GTAC_CONFIG.Option_Robot_Count<6) AND
											(MAIN.R7.Task_ID_Ack=Brake_Test AND MAIN.R7.Operating OR GTAC_CONFIG.Option_Robot_Count<7) AND
											(MAIN.R8.Task_ID_Ack=Brake_Test AND MAIN.R8.Operating OR GTAC_CONFIG.Option_Robot_Count<8) AND
											(MAIN.R9.Task_ID_Ack=Brake_Test AND MAIN.R9.Operating OR GTAC_CONFIG.Option_Robot_Count<9) AND
											(MAIN.R10.Task_ID_Ack=Brake_Test AND MAIN.R10.Operating OR GTAC_CONFIG.Option_Robot_Count<10) AND
											(MAIN.R11.Task_ID_Ack=Brake_Test AND MAIN.R11.Operating OR GTAC_CONFIG.Option_Robot_Count<11) AND
											(MAIN.R12.Task_ID_Ack=Brake_Test AND MAIN.R12.Operating OR GTAC_CONFIG.Option_Robot_Count<12) AND
											(MAIN.R13.Task_ID_Ack=Brake_Test AND MAIN.R13.Operating OR GTAC_CONFIG.Option_Robot_Count<13) AND
											(MAIN.R14.Task_ID_Ack=Brake_Test AND MAIN.R14.Operating OR GTAC_CONFIG.Option_Robot_Count<14) AND
											(MAIN.R15.Task_ID_Ack=Brake_Test AND MAIN.R15.Operating OR GTAC_CONFIG.Option_Robot_Count<15) AND
											(MAIN.R16.Task_ID_Ack=Brake_Test AND MAIN.R16.Operating OR GTAC_CONFIG.Option_Robot_Count<16) AND
											(MAIN.R17.Task_ID_Ack=Brake_Test AND MAIN.R17.Operating OR GTAC_CONFIG.Option_Robot_Count<17) AND
											(MAIN.R18.Task_ID_Ack=Brake_Test AND MAIN.R18.Operating OR GTAC_CONFIG.Option_Robot_Count<18) AND
											(MAIN.R19.Task_ID_Ack=Brake_Test AND MAIN.R19.Operating OR GTAC_CONFIG.Option_Robot_Count<19) AND
											(MAIN.R20.Task_ID_Ack=Brake_Test AND MAIN.R20.Operating OR GTAC_CONFIG.Option_Robot_Count<20) AND
											(MAIN.R21.Task_ID_Ack=Brake_Test AND MAIN.R21.Operating OR GTAC_CONFIG.Option_Robot_Count<21) AND
											(MAIN.R22.Task_ID_Ack=Brake_Test AND MAIN.R22.Operating OR GTAC_CONFIG.Option_Robot_Count<22) AND
											(MAIN.R23.Task_ID_Ack=Brake_Test AND MAIN.R23.Operating OR GTAC_CONFIG.Option_Robot_Count<23) AND
											(MAIN.R24.Task_ID_Ack=Brake_Test AND MAIN.R24.Operating OR GTAC_CONFIG.Option_Robot_Count<24) AND
											(MAIN.R25.Task_ID_Ack=Brake_Test AND MAIN.R25.Operating OR GTAC_CONFIG.Option_Robot_Count<25) AND
											(MAIN.R26.Task_ID_Ack=Brake_Test AND MAIN.R26.Operating OR GTAC_CONFIG.Option_Robot_Count<26) AND
											(MAIN.R27.Task_ID_Ack=Brake_Test AND MAIN.R27.Operating OR GTAC_CONFIG.Option_Robot_Count<27) AND
											(MAIN.R28.Task_ID_Ack=Brake_Test AND MAIN.R28.Operating OR GTAC_CONFIG.Option_Robot_Count<28) AND
											(MAIN.R29.Task_ID_Ack=Brake_Test AND MAIN.R29.Operating OR GTAC_CONFIG.Option_Robot_Count<29) AND
											(MAIN.R30.Task_ID_Ack=Brake_Test AND MAIN.R30.Operating OR GTAC_CONFIG.Option_Robot_Count<30))
											OR
							(Start_All_TCRobots AND MAIN.R1.Task_ID_Ack=Tip_Change AND MAIN.R1.Operating AND
											(MAIN.R2.Task_ID_Ack=Tip_Change AND MAIN.R2.Operating OR GTAC_CONFIG.Option_Robot_Count<2) AND
											(MAIN.R3.Task_ID_Ack=Tip_Change AND MAIN.R3.Operating OR GTAC_CONFIG.Option_Robot_Count<3) AND
											(MAIN.R4.Task_ID_Ack=Tip_Change AND MAIN.R4.Operating OR GTAC_CONFIG.Option_Robot_Count<4) AND
											(MAIN.R5.Task_ID_Ack=Tip_Change AND MAIN.R5.Operating OR GTAC_CONFIG.Option_Robot_Count<5) AND
											(MAIN.R6.Task_ID_Ack=Tip_Change AND MAIN.R6.Operating OR GTAC_CONFIG.Option_Robot_Count<6) AND
											(MAIN.R7.Task_ID_Ack=Tip_Change AND MAIN.R7.Operating OR GTAC_CONFIG.Option_Robot_Count<7) AND
											(MAIN.R8.Task_ID_Ack=Tip_Change AND MAIN.R8.Operating OR GTAC_CONFIG.Option_Robot_Count<8) AND
											(MAIN.R9.Task_ID_Ack=Tip_Change AND MAIN.R9.Operating OR GTAC_CONFIG.Option_Robot_Count<9) AND
											(MAIN.R10.Task_ID_Ack=Tip_Change AND MAIN.R10.Operating OR GTAC_CONFIG.Option_Robot_Count<10) AND
											(MAIN.R11.Task_ID_Ack=Tip_Change AND MAIN.R11.Operating OR GTAC_CONFIG.Option_Robot_Count<11) AND
											(MAIN.R12.Task_ID_Ack=Tip_Change AND MAIN.R12.Operating OR GTAC_CONFIG.Option_Robot_Count<12) AND
											(MAIN.R13.Task_ID_Ack=Tip_Change AND MAIN.R13.Operating OR GTAC_CONFIG.Option_Robot_Count<13) AND
											(MAIN.R14.Task_ID_Ack=Tip_Change AND MAIN.R14.Operating OR GTAC_CONFIG.Option_Robot_Count<14) AND
											(MAIN.R15.Task_ID_Ack=Tip_Change AND MAIN.R15.Operating OR GTAC_CONFIG.Option_Robot_Count<15) AND
											(MAIN.R16.Task_ID_Ack=Tip_Change AND MAIN.R16.Operating OR GTAC_CONFIG.Option_Robot_Count<16) AND
											(MAIN.R17.Task_ID_Ack=Tip_Change AND MAIN.R17.Operating OR GTAC_CONFIG.Option_Robot_Count<17) AND
											(MAIN.R18.Task_ID_Ack=Tip_Change AND MAIN.R18.Operating OR GTAC_CONFIG.Option_Robot_Count<18) AND
											(MAIN.R19.Task_ID_Ack=Tip_Change AND MAIN.R19.Operating OR GTAC_CONFIG.Option_Robot_Count<19) AND
											(MAIN.R20.Task_ID_Ack=Tip_Change AND MAIN.R20.Operating OR GTAC_CONFIG.Option_Robot_Count<20) AND
											(MAIN.R21.Task_ID_Ack=Tip_Change AND MAIN.R21.Operating OR GTAC_CONFIG.Option_Robot_Count<21) AND
											(MAIN.R22.Task_ID_Ack=Tip_Change AND MAIN.R22.Operating OR GTAC_CONFIG.Option_Robot_Count<22) AND
											(MAIN.R23.Task_ID_Ack=Tip_Change AND MAIN.R23.Operating OR GTAC_CONFIG.Option_Robot_Count<23) AND
											(MAIN.R24.Task_ID_Ack=Tip_Change AND MAIN.R24.Operating OR GTAC_CONFIG.Option_Robot_Count<24) AND
											(MAIN.R25.Task_ID_Ack=Tip_Change AND MAIN.R25.Operating OR GTAC_CONFIG.Option_Robot_Count<25) AND
											(MAIN.R26.Task_ID_Ack=Tip_Change AND MAIN.R26.Operating OR GTAC_CONFIG.Option_Robot_Count<26) AND
											(MAIN.R27.Task_ID_Ack=Tip_Change AND MAIN.R27.Operating OR GTAC_CONFIG.Option_Robot_Count<27) AND
											(MAIN.R28.Task_ID_Ack=Tip_Change AND MAIN.R28.Operating OR GTAC_CONFIG.Option_Robot_Count<28) AND
											(MAIN.R29.Task_ID_Ack=Tip_Change AND MAIN.R29.Operating OR GTAC_CONFIG.Option_Robot_Count<29) AND
											(MAIN.R30.Task_ID_Ack=Tip_Change AND MAIN.R30.Operating OR GTAC_CONFIG.Option_Robot_Count<30))
											OR
							(Start_All_TDRobots AND MAIN.R1.Task_ID_Ack=Tip_Dress AND MAIN.R1.Operating AND
											(MAIN.R2.Task_ID_Ack=Tip_Dress AND MAIN.R2.Operating OR GTAC_CONFIG.Option_Robot_Count<2) AND
											(MAIN.R3.Task_ID_Ack=Tip_Dress AND MAIN.R3.Operating OR GTAC_CONFIG.Option_Robot_Count<3) AND
											(MAIN.R4.Task_ID_Ack=Tip_Dress AND MAIN.R4.Operating OR GTAC_CONFIG.Option_Robot_Count<4) AND
											(MAIN.R5.Task_ID_Ack=Tip_Dress AND MAIN.R5.Operating OR GTAC_CONFIG.Option_Robot_Count<5) AND
											(MAIN.R6.Task_ID_Ack=Tip_Dress AND MAIN.R6.Operating OR GTAC_CONFIG.Option_Robot_Count<6) AND
											(MAIN.R7.Task_ID_Ack=Tip_Dress AND MAIN.R7.Operating OR GTAC_CONFIG.Option_Robot_Count<7) AND
											(MAIN.R8.Task_ID_Ack=Tip_Dress AND MAIN.R8.Operating OR GTAC_CONFIG.Option_Robot_Count<8) AND
											(MAIN.R9.Task_ID_Ack=Tip_Dress AND MAIN.R9.Operating OR GTAC_CONFIG.Option_Robot_Count<9) AND
											(MAIN.R10.Task_ID_Ack=Tip_Dress AND MAIN.R10.Operating OR GTAC_CONFIG.Option_Robot_Count<10) AND
											(MAIN.R11.Task_ID_Ack=Tip_Dress AND MAIN.R11.Operating OR GTAC_CONFIG.Option_Robot_Count<11) AND
											(MAIN.R12.Task_ID_Ack=Tip_Dress AND MAIN.R12.Operating OR GTAC_CONFIG.Option_Robot_Count<12) AND
											(MAIN.R13.Task_ID_Ack=Tip_Dress AND MAIN.R13.Operating OR GTAC_CONFIG.Option_Robot_Count<13) AND
											(MAIN.R14.Task_ID_Ack=Tip_Dress AND MAIN.R14.Operating OR GTAC_CONFIG.Option_Robot_Count<14) AND
											(MAIN.R15.Task_ID_Ack=Tip_Dress AND MAIN.R15.Operating OR GTAC_CONFIG.Option_Robot_Count<15) AND
											(MAIN.R16.Task_ID_Ack=Tip_Dress AND MAIN.R16.Operating OR GTAC_CONFIG.Option_Robot_Count<16) AND
											(MAIN.R17.Task_ID_Ack=Tip_Dress AND MAIN.R17.Operating OR GTAC_CONFIG.Option_Robot_Count<17) AND
											(MAIN.R18.Task_ID_Ack=Tip_Dress AND MAIN.R18.Operating OR GTAC_CONFIG.Option_Robot_Count<18) AND
											(MAIN.R19.Task_ID_Ack=Tip_Dress AND MAIN.R19.Operating OR GTAC_CONFIG.Option_Robot_Count<19) AND
											(MAIN.R20.Task_ID_Ack=Tip_Dress AND MAIN.R20.Operating OR GTAC_CONFIG.Option_Robot_Count<20) AND
											(MAIN.R21.Task_ID_Ack=Tip_Dress AND MAIN.R21.Operating OR GTAC_CONFIG.Option_Robot_Count<21) AND
											(MAIN.R22.Task_ID_Ack=Tip_Dress AND MAIN.R22.Operating OR GTAC_CONFIG.Option_Robot_Count<22) AND
											(MAIN.R23.Task_ID_Ack=Tip_Dress AND MAIN.R23.Operating OR GTAC_CONFIG.Option_Robot_Count<23) AND
											(MAIN.R24.Task_ID_Ack=Tip_Dress AND MAIN.R24.Operating OR GTAC_CONFIG.Option_Robot_Count<24) AND
											(MAIN.R25.Task_ID_Ack=Tip_Dress AND MAIN.R25.Operating OR GTAC_CONFIG.Option_Robot_Count<25) AND
											(MAIN.R26.Task_ID_Ack=Tip_Dress AND MAIN.R26.Operating OR GTAC_CONFIG.Option_Robot_Count<26) AND
											(MAIN.R27.Task_ID_Ack=Tip_Dress AND MAIN.R27.Operating OR GTAC_CONFIG.Option_Robot_Count<27) AND
											(MAIN.R28.Task_ID_Ack=Tip_Dress AND MAIN.R28.Operating OR GTAC_CONFIG.Option_Robot_Count<28) AND
											(MAIN.R29.Task_ID_Ack=Tip_Dress AND MAIN.R29.Operating OR GTAC_CONFIG.Option_Robot_Count<29) AND
											(MAIN.R30.Task_ID_Ack=Tip_Dress AND MAIN.R30.Operating OR GTAC_CONFIG.Option_Robot_Count<30))
											OR
							(Start_All_TraccTCP AND MAIN.R1.Task_ID_Ack=Tracc_TCP AND MAIN.R1.Operating AND
											(MAIN.R2.Task_ID_Ack=Tracc_TCP AND MAIN.R2.Operating OR GTAC_CONFIG.Option_Robot_Count<2) AND
											(MAIN.R3.Task_ID_Ack=Tracc_TCP AND MAIN.R3.Operating OR GTAC_CONFIG.Option_Robot_Count<3) AND
											(MAIN.R4.Task_ID_Ack=Tracc_TCP AND MAIN.R4.Operating OR GTAC_CONFIG.Option_Robot_Count<4) AND
											(MAIN.R5.Task_ID_Ack=Tracc_TCP AND MAIN.R5.Operating OR GTAC_CONFIG.Option_Robot_Count<5) AND
											(MAIN.R6.Task_ID_Ack=Tracc_TCP AND MAIN.R6.Operating OR GTAC_CONFIG.Option_Robot_Count<6) AND
											(MAIN.R7.Task_ID_Ack=Tracc_TCP AND MAIN.R7.Operating OR GTAC_CONFIG.Option_Robot_Count<7) AND
											(MAIN.R8.Task_ID_Ack=Tracc_TCP AND MAIN.R8.Operating OR GTAC_CONFIG.Option_Robot_Count<8) AND
											(MAIN.R9.Task_ID_Ack=Tracc_TCP AND MAIN.R9.Operating OR GTAC_CONFIG.Option_Robot_Count<9) AND
											(MAIN.R10.Task_ID_Ack=Tracc_TCP AND MAIN.R10.Operating OR GTAC_CONFIG.Option_Robot_Count<10) AND
											(MAIN.R11.Task_ID_Ack=Tracc_TCP AND MAIN.R11.Operating OR GTAC_CONFIG.Option_Robot_Count<11) AND
											(MAIN.R12.Task_ID_Ack=Tracc_TCP AND MAIN.R12.Operating OR GTAC_CONFIG.Option_Robot_Count<12) AND
											(MAIN.R13.Task_ID_Ack=Tracc_TCP AND MAIN.R13.Operating OR GTAC_CONFIG.Option_Robot_Count<13) AND
											(MAIN.R14.Task_ID_Ack=Tracc_TCP AND MAIN.R14.Operating OR GTAC_CONFIG.Option_Robot_Count<14) AND
											(MAIN.R15.Task_ID_Ack=Tracc_TCP AND MAIN.R15.Operating OR GTAC_CONFIG.Option_Robot_Count<15) AND
											(MAIN.R16.Task_ID_Ack=Tracc_TCP AND MAIN.R16.Operating OR GTAC_CONFIG.Option_Robot_Count<16) AND
											(MAIN.R17.Task_ID_Ack=Tracc_TCP AND MAIN.R17.Operating OR GTAC_CONFIG.Option_Robot_Count<17) AND
											(MAIN.R18.Task_ID_Ack=Tracc_TCP AND MAIN.R18.Operating OR GTAC_CONFIG.Option_Robot_Count<18) AND
											(MAIN.R19.Task_ID_Ack=Tracc_TCP AND MAIN.R19.Operating OR GTAC_CONFIG.Option_Robot_Count<19) AND
											(MAIN.R20.Task_ID_Ack=Tracc_TCP AND MAIN.R20.Operating OR GTAC_CONFIG.Option_Robot_Count<20) AND
											(MAIN.R21.Task_ID_Ack=Tracc_TCP AND MAIN.R21.Operating OR GTAC_CONFIG.Option_Robot_Count<21) AND
											(MAIN.R22.Task_ID_Ack=Tracc_TCP AND MAIN.R22.Operating OR GTAC_CONFIG.Option_Robot_Count<22) AND
											(MAIN.R23.Task_ID_Ack=Tracc_TCP AND MAIN.R23.Operating OR GTAC_CONFIG.Option_Robot_Count<23) AND
											(MAIN.R24.Task_ID_Ack=Tracc_TCP AND MAIN.R24.Operating OR GTAC_CONFIG.Option_Robot_Count<24) AND
											(MAIN.R25.Task_ID_Ack=Tracc_TCP AND MAIN.R25.Operating OR GTAC_CONFIG.Option_Robot_Count<25) AND
											(MAIN.R26.Task_ID_Ack=Tracc_TCP AND MAIN.R26.Operating OR GTAC_CONFIG.Option_Robot_Count<26) AND
											(MAIN.R27.Task_ID_Ack=Tracc_TCP AND MAIN.R27.Operating OR GTAC_CONFIG.Option_Robot_Count<27) AND
											(MAIN.R28.Task_ID_Ack=Tracc_TCP AND MAIN.R28.Operating OR GTAC_CONFIG.Option_Robot_Count<28) AND
											(MAIN.R29.Task_ID_Ack=Tracc_TCP AND MAIN.R29.Operating OR GTAC_CONFIG.Option_Robot_Count<29) AND
											(MAIN.R30.Task_ID_Ack=Tracc_TCP AND MAIN.R30.Operating OR GTAC_CONFIG.Option_Robot_Count<30));
		All_Robots_Complete:= (Start_All_MTRobots AND MAIN.R1.Task_ID_Ack=Master_Test AND MAIN.R1.Task_Completed AND
											(MAIN.R2.Task_ID_Ack=Master_Test AND MAIN.R2.Task_Completed OR GTAC_CONFIG.Option_Robot_Count<2) AND
											(MAIN.R3.Task_ID_Ack=Master_Test AND MAIN.R3.Task_Completed OR GTAC_CONFIG.Option_Robot_Count<3) AND
											(MAIN.R4.Task_ID_Ack=Master_Test AND MAIN.R4.Task_Completed OR GTAC_CONFIG.Option_Robot_Count<4) AND
											(MAIN.R5.Task_ID_Ack=Master_Test AND MAIN.R5.Task_Completed OR GTAC_CONFIG.Option_Robot_Count<5) AND
											(MAIN.R6.Task_ID_Ack=Master_Test AND MAIN.R6.Task_Completed OR GTAC_CONFIG.Option_Robot_Count<6) AND
											(MAIN.R7.Task_ID_Ack=Master_Test AND MAIN.R7.Task_Completed OR GTAC_CONFIG.Option_Robot_Count<7) AND
											(MAIN.R8.Task_ID_Ack= Master_Test AND MAIN.R8.Task_Completed OR GTAC_CONFIG.Option_Robot_Count<8) AND
											(MAIN.R9.Task_ID_Ack=Master_Test AND MAIN.R9.Task_Completed OR GTAC_CONFIG.Option_Robot_Count<9) AND
											(MAIN.R10.Task_ID_Ack=Master_Test AND MAIN.R10.Task_Completed OR GTAC_CONFIG.Option_Robot_Count<10) AND
											(MAIN.R11.Task_ID_Ack=Master_Test AND MAIN.R11.Task_Completed OR GTAC_CONFIG.Option_Robot_Count<11) AND
											(MAIN.R12.Task_ID_Ack=Master_Test AND MAIN.R12.Task_Completed OR GTAC_CONFIG.Option_Robot_Count<12) AND
											(MAIN.R13.Task_ID_Ack=Master_Test AND MAIN.R13.Task_Completed OR GTAC_CONFIG.Option_Robot_Count<13) AND
											(MAIN.R14.Task_ID_Ack=Master_Test AND MAIN.R14.Task_Completed OR GTAC_CONFIG.Option_Robot_Count<14) AND
											(MAIN.R15.Task_ID_Ack=Master_Test AND MAIN.R15.Task_Completed OR GTAC_CONFIG.Option_Robot_Count<15) AND
											(MAIN.R16.Task_ID_Ack=Master_Test AND MAIN.R16.Task_Completed OR GTAC_CONFIG.Option_Robot_Count<16) AND
											(MAIN.R17.Task_ID_Ack=Master_Test AND MAIN.R17.Task_Completed OR GTAC_CONFIG.Option_Robot_Count<17) AND
											(MAIN.R18.Task_ID_Ack= Master_Test AND MAIN.R18.Task_Completed OR GTAC_CONFIG.Option_Robot_Count<18) AND
											(MAIN.R19.Task_ID_Ack=Master_Test AND MAIN.R19.Task_Completed OR GTAC_CONFIG.Option_Robot_Count<19) AND
											(MAIN.R20.Task_ID_Ack=Master_Test AND MAIN.R20.Task_Completed OR GTAC_CONFIG.Option_Robot_Count<20) AND
											(MAIN.R21.Task_ID_Ack=Master_Test AND MAIN.R21.Task_Completed OR GTAC_CONFIG.Option_Robot_Count<21) AND
											(MAIN.R22.Task_ID_Ack=Master_Test AND MAIN.R22.Task_Completed OR GTAC_CONFIG.Option_Robot_Count<22) AND
											(MAIN.R23.Task_ID_Ack=Master_Test AND MAIN.R23.Task_Completed OR GTAC_CONFIG.Option_Robot_Count<23) AND
											(MAIN.R24.Task_ID_Ack=Master_Test AND MAIN.R24.Task_Completed OR GTAC_CONFIG.Option_Robot_Count<24) AND
											(MAIN.R25.Task_ID_Ack=Master_Test AND MAIN.R25.Task_Completed OR GTAC_CONFIG.Option_Robot_Count<25) AND
											(MAIN.R26.Task_ID_Ack=Master_Test AND MAIN.R26.Task_Completed OR GTAC_CONFIG.Option_Robot_Count<26) AND
											(MAIN.R27.Task_ID_Ack=Master_Test AND MAIN.R27.Task_Completed OR GTAC_CONFIG.Option_Robot_Count<27) AND
											(MAIN.R28.Task_ID_Ack=Master_Test AND MAIN.R28.Task_Completed OR GTAC_CONFIG.Option_Robot_Count<28) AND
											(MAIN.R29.Task_ID_Ack=Master_Test AND MAIN.R29.Task_Completed OR GTAC_CONFIG.Option_Robot_Count<29) AND
											(MAIN.R30.Task_ID_Ack=Master_Test AND MAIN.R30.Task_Completed OR GTAC_CONFIG.Option_Robot_Count<30))
											OR
							(Start_All_BTRobots AND MAIN.R1.Task_ID_Ack=Brake_Test AND MAIN.R1.Task_Completed AND
											(MAIN.R2.Task_ID_Ack=Brake_Test AND MAIN.R2.Task_Completed OR GTAC_CONFIG.Option_Robot_Count<2) AND
											(MAIN.R3.Task_ID_Ack=Brake_Test AND MAIN.R3.Task_Completed OR GTAC_CONFIG.Option_Robot_Count<3) AND
											(MAIN.R4.Task_ID_Ack=Brake_Test AND MAIN.R4.Task_Completed OR GTAC_CONFIG.Option_Robot_Count<4) AND
											(MAIN.R5.Task_ID_Ack=Brake_Test AND MAIN.R5.Task_Completed OR GTAC_CONFIG.Option_Robot_Count<5) AND
											(MAIN.R6.Task_ID_Ack=Brake_Test AND MAIN.R6.Task_Completed OR GTAC_CONFIG.Option_Robot_Count<6) AND
											(MAIN.R7.Task_ID_Ack=Brake_Test AND MAIN.R7.Task_Completed OR GTAC_CONFIG.Option_Robot_Count<7) AND
											(MAIN.R8.Task_ID_Ack=Brake_Test AND MAIN.R8.Task_Completed OR GTAC_CONFIG.Option_Robot_Count<8) AND
											(MAIN.R9.Task_ID_Ack=Brake_Test AND MAIN.R9.Task_Completed OR GTAC_CONFIG.Option_Robot_Count<9) AND
											(MAIN.R10.Task_ID_Ack=Brake_Test AND MAIN.R10.Task_Completed OR GTAC_CONFIG.Option_Robot_Count<10) AND
											(MAIN.R11.Task_ID_Ack=Brake_Test AND MAIN.R11.Task_Completed OR GTAC_CONFIG.Option_Robot_Count<11) AND
											(MAIN.R12.Task_ID_Ack=Brake_Test AND MAIN.R12.Task_Completed OR GTAC_CONFIG.Option_Robot_Count<12) AND
											(MAIN.R13.Task_ID_Ack=Brake_Test AND MAIN.R13.Task_Completed OR GTAC_CONFIG.Option_Robot_Count<13) AND
											(MAIN.R14.Task_ID_Ack=Brake_Test AND MAIN.R14.Task_Completed OR GTAC_CONFIG.Option_Robot_Count<14) AND
											(MAIN.R15.Task_ID_Ack=Brake_Test AND MAIN.R15.Task_Completed OR GTAC_CONFIG.Option_Robot_Count<15) AND
											(MAIN.R16.Task_ID_Ack=Brake_Test AND MAIN.R16.Task_Completed OR GTAC_CONFIG.Option_Robot_Count<16) AND
											(MAIN.R17.Task_ID_Ack=Brake_Test AND MAIN.R17.Task_Completed OR GTAC_CONFIG.Option_Robot_Count<17) AND
											(MAIN.R18.Task_ID_Ack=Brake_Test AND MAIN.R18.Task_Completed OR GTAC_CONFIG.Option_Robot_Count<18) AND
											(MAIN.R19.Task_ID_Ack=Brake_Test AND MAIN.R19.Task_Completed OR GTAC_CONFIG.Option_Robot_Count<19) AND
											(MAIN.R20.Task_ID_Ack=Brake_Test AND MAIN.R20.Task_Completed OR GTAC_CONFIG.Option_Robot_Count<20) AND
											(MAIN.R21.Task_ID_Ack=Brake_Test AND MAIN.R21.Task_Completed OR GTAC_CONFIG.Option_Robot_Count<21) AND
											(MAIN.R22.Task_ID_Ack=Brake_Test AND MAIN.R22.Task_Completed OR GTAC_CONFIG.Option_Robot_Count<22) AND
											(MAIN.R23.Task_ID_Ack=Brake_Test AND MAIN.R23.Task_Completed OR GTAC_CONFIG.Option_Robot_Count<23) AND
											(MAIN.R24.Task_ID_Ack=Brake_Test AND MAIN.R24.Task_Completed OR GTAC_CONFIG.Option_Robot_Count<24) AND
											(MAIN.R25.Task_ID_Ack=Brake_Test AND MAIN.R25.Task_Completed OR GTAC_CONFIG.Option_Robot_Count<25) AND
											(MAIN.R26.Task_ID_Ack=Brake_Test AND MAIN.R26.Task_Completed OR GTAC_CONFIG.Option_Robot_Count<26) AND
											(MAIN.R27.Task_ID_Ack=Brake_Test AND MAIN.R27.Task_Completed OR GTAC_CONFIG.Option_Robot_Count<27) AND
											(MAIN.R28.Task_ID_Ack=Brake_Test AND MAIN.R28.Task_Completed OR GTAC_CONFIG.Option_Robot_Count<28) AND
											(MAIN.R29.Task_ID_Ack=Brake_Test AND MAIN.R29.Task_Completed OR GTAC_CONFIG.Option_Robot_Count<29) AND
											(MAIN.R30.Task_ID_Ack=Brake_Test AND MAIN.R30.Task_Completed OR GTAC_CONFIG.Option_Robot_Count<30))
											OR
							(Start_All_TCRobots AND MAIN.R1.Task_ID_Ack=Tip_Change AND MAIN.R1.Task_Completed AND
											(MAIN.R2.Task_ID_Ack=Tip_Change AND MAIN.R2.Task_Completed OR GTAC_CONFIG.Option_Robot_Count<2) AND
											(MAIN.R3.Task_ID_Ack=Tip_Change AND MAIN.R3.Task_Completed OR GTAC_CONFIG.Option_Robot_Count<3) AND
											(MAIN.R4.Task_ID_Ack=Tip_Change AND MAIN.R4.Task_Completed OR GTAC_CONFIG.Option_Robot_Count<4) AND
											(MAIN.R5.Task_ID_Ack=Tip_Change AND MAIN.R5.Task_Completed OR GTAC_CONFIG.Option_Robot_Count<5) AND
											(MAIN.R6.Task_ID_Ack=Tip_Change AND MAIN.R6.Task_Completed OR GTAC_CONFIG.Option_Robot_Count<6) AND
											(MAIN.R7.Task_ID_Ack=Tip_Change AND MAIN.R7.Task_Completed OR GTAC_CONFIG.Option_Robot_Count<7) AND
											(MAIN.R8.Task_ID_Ack=Tip_Change AND MAIN.R8.Task_Completed OR GTAC_CONFIG.Option_Robot_Count<8) AND
											(MAIN.R9.Task_ID_Ack=Tip_Change AND MAIN.R9.Task_Completed OR GTAC_CONFIG.Option_Robot_Count<9) AND
											(MAIN.R10.Task_ID_Ack=Tip_Change AND MAIN.R10.Task_Completed OR GTAC_CONFIG.Option_Robot_Count<10) AND
											(MAIN.R11.Task_ID_Ack=Tip_Change AND MAIN.R11.Task_Completed OR GTAC_CONFIG.Option_Robot_Count<11) AND
											(MAIN.R12.Task_ID_Ack=Tip_Change AND MAIN.R12.Task_Completed OR GTAC_CONFIG.Option_Robot_Count<12) AND
											(MAIN.R13.Task_ID_Ack=Tip_Change AND MAIN.R13.Task_Completed OR GTAC_CONFIG.Option_Robot_Count<13) AND
											(MAIN.R14.Task_ID_Ack=Tip_Change AND MAIN.R14.Task_Completed OR GTAC_CONFIG.Option_Robot_Count<14) AND
											(MAIN.R15.Task_ID_Ack=Tip_Change AND MAIN.R15.Task_Completed OR GTAC_CONFIG.Option_Robot_Count<15) AND
											(MAIN.R16.Task_ID_Ack=Tip_Change AND MAIN.R16.Task_Completed OR GTAC_CONFIG.Option_Robot_Count<16) AND
											(MAIN.R17.Task_ID_Ack=Tip_Change AND MAIN.R17.Task_Completed OR GTAC_CONFIG.Option_Robot_Count<17) AND
											(MAIN.R18.Task_ID_Ack=Tip_Change AND MAIN.R18.Task_Completed OR GTAC_CONFIG.Option_Robot_Count<18) AND
											(MAIN.R19.Task_ID_Ack=Tip_Change AND MAIN.R19.Task_Completed OR GTAC_CONFIG.Option_Robot_Count<19) AND
											(MAIN.R20.Task_ID_Ack=Tip_Change AND MAIN.R20.Task_Completed OR GTAC_CONFIG.Option_Robot_Count<20) AND
											(MAIN.R21.Task_ID_Ack=Tip_Change AND MAIN.R21.Task_Completed OR GTAC_CONFIG.Option_Robot_Count<21) AND
											(MAIN.R22.Task_ID_Ack=Tip_Change AND MAIN.R22.Task_Completed OR GTAC_CONFIG.Option_Robot_Count<22) AND
											(MAIN.R23.Task_ID_Ack=Tip_Change AND MAIN.R23.Task_Completed OR GTAC_CONFIG.Option_Robot_Count<23) AND
											(MAIN.R24.Task_ID_Ack=Tip_Change AND MAIN.R24.Task_Completed OR GTAC_CONFIG.Option_Robot_Count<24) AND
											(MAIN.R25.Task_ID_Ack=Tip_Change AND MAIN.R25.Task_Completed OR GTAC_CONFIG.Option_Robot_Count<25) AND
											(MAIN.R26.Task_ID_Ack=Tip_Change AND MAIN.R26.Task_Completed OR GTAC_CONFIG.Option_Robot_Count<26) AND
											(MAIN.R27.Task_ID_Ack=Tip_Change AND MAIN.R27.Task_Completed OR GTAC_CONFIG.Option_Robot_Count<27) AND
											(MAIN.R28.Task_ID_Ack=Tip_Change AND MAIN.R28.Task_Completed OR GTAC_CONFIG.Option_Robot_Count<28) AND
											(MAIN.R29.Task_ID_Ack=Tip_Change AND MAIN.R29.Task_Completed OR GTAC_CONFIG.Option_Robot_Count<29) AND
											(MAIN.R30.Task_ID_Ack=Tip_Change AND MAIN.R30.Task_Completed OR GTAC_CONFIG.Option_Robot_Count<30) AND
											All_Robots_SteppersRST)
											OR
							(Start_All_TDRobots AND MAIN.R1.Task_ID_Ack=Tip_Dress AND MAIN.R1.Task_Completed AND
											(MAIN.R2.Task_ID_Ack=Tip_Dress AND MAIN.R2.Task_Completed OR GTAC_CONFIG.Option_Robot_Count<2) AND
											(MAIN.R3.Task_ID_Ack=Tip_Dress AND MAIN.R3.Task_Completed OR GTAC_CONFIG.Option_Robot_Count<3) AND
											(MAIN.R4.Task_ID_Ack=Tip_Dress AND MAIN.R4.Task_Completed OR GTAC_CONFIG.Option_Robot_Count<4) AND
											(MAIN.R5.Task_ID_Ack=Tip_Dress AND MAIN.R5.Task_Completed OR GTAC_CONFIG.Option_Robot_Count<5) AND
											(MAIN.R6.Task_ID_Ack=Tip_Dress AND MAIN.R6.Task_Completed OR GTAC_CONFIG.Option_Robot_Count<6) AND
											(MAIN.R7.Task_ID_Ack=Tip_Dress AND MAIN.R7.Task_Completed OR GTAC_CONFIG.Option_Robot_Count<7) AND
											(MAIN.R8.Task_ID_Ack=Tip_Dress AND MAIN.R8.Task_Completed OR GTAC_CONFIG.Option_Robot_Count<8) AND
											(MAIN.R9.Task_ID_Ack=Tip_Dress AND MAIN.R9.Task_Completed OR GTAC_CONFIG.Option_Robot_Count<9) AND
											(MAIN.R10.Task_ID_Ack=Tip_Dress AND MAIN.R10.Task_Completed OR GTAC_CONFIG.Option_Robot_Count<10) AND
											(MAIN.R11.Task_ID_Ack=Tip_Dress AND MAIN.R11.Task_Completed OR GTAC_CONFIG.Option_Robot_Count<11) AND
											(MAIN.R12.Task_ID_Ack=Tip_Dress AND MAIN.R12.Task_Completed OR GTAC_CONFIG.Option_Robot_Count<12) AND
											(MAIN.R13.Task_ID_Ack=Tip_Dress AND MAIN.R13.Task_Completed OR GTAC_CONFIG.Option_Robot_Count<13) AND
											(MAIN.R14.Task_ID_Ack=Tip_Dress AND MAIN.R14.Task_Completed OR GTAC_CONFIG.Option_Robot_Count<14) AND
											(MAIN.R15.Task_ID_Ack=Tip_Dress AND MAIN.R15.Task_Completed OR GTAC_CONFIG.Option_Robot_Count<15) AND
											(MAIN.R16.Task_ID_Ack=Tip_Dress AND MAIN.R16.Task_Completed OR GTAC_CONFIG.Option_Robot_Count<16) AND
											(MAIN.R17.Task_ID_Ack=Tip_Dress AND MAIN.R17.Task_Completed OR GTAC_CONFIG.Option_Robot_Count<17) AND
											(MAIN.R18.Task_ID_Ack=Tip_Dress AND MAIN.R18.Task_Completed OR GTAC_CONFIG.Option_Robot_Count<18) AND
											(MAIN.R19.Task_ID_Ack=Tip_Dress AND MAIN.R19.Task_Completed OR GTAC_CONFIG.Option_Robot_Count<19) AND
											(MAIN.R20.Task_ID_Ack=Tip_Dress AND MAIN.R20.Task_Completed OR GTAC_CONFIG.Option_Robot_Count<20) AND
											(MAIN.R21.Task_ID_Ack=Tip_Dress AND MAIN.R21.Task_Completed OR GTAC_CONFIG.Option_Robot_Count<21) AND
											(MAIN.R22.Task_ID_Ack=Tip_Dress AND MAIN.R22.Task_Completed OR GTAC_CONFIG.Option_Robot_Count<22) AND
											(MAIN.R23.Task_ID_Ack=Tip_Dress AND MAIN.R23.Task_Completed OR GTAC_CONFIG.Option_Robot_Count<23) AND
											(MAIN.R24.Task_ID_Ack=Tip_Dress AND MAIN.R24.Task_Completed OR GTAC_CONFIG.Option_Robot_Count<24) AND
											(MAIN.R25.Task_ID_Ack=Tip_Dress AND MAIN.R25.Task_Completed OR GTAC_CONFIG.Option_Robot_Count<25) AND
											(MAIN.R26.Task_ID_Ack=Tip_Dress AND MAIN.R26.Task_Completed OR GTAC_CONFIG.Option_Robot_Count<26) AND
											(MAIN.R27.Task_ID_Ack=Tip_Dress AND MAIN.R27.Task_Completed OR GTAC_CONFIG.Option_Robot_Count<27) AND
											(MAIN.R28.Task_ID_Ack=Tip_Dress AND MAIN.R28.Task_Completed OR GTAC_CONFIG.Option_Robot_Count<28) AND
											(MAIN.R29.Task_ID_Ack=Tip_Dress AND MAIN.R29.Task_Completed OR GTAC_CONFIG.Option_Robot_Count<29) AND
											(MAIN.R30.Task_ID_Ack=Tip_Dress AND MAIN.R30.Task_Completed OR GTAC_CONFIG.Option_Robot_Count<30))
											OR
							(Start_All_TraccTCP AND MAIN.R1.Task_ID_Ack=Tracc_TCP AND MAIN.R1.Task_Completed AND
											(MAIN.R2.Task_ID_Ack=Tracc_TCP AND MAIN.R2.Task_Completed OR GTAC_CONFIG.Option_Robot_Count<2) AND
											(MAIN.R3.Task_ID_Ack=Tracc_TCP AND MAIN.R3.Task_Completed OR GTAC_CONFIG.Option_Robot_Count<3) AND
											(MAIN.R4.Task_ID_Ack=Tracc_TCP AND MAIN.R4.Task_Completed OR GTAC_CONFIG.Option_Robot_Count<4) AND
											(MAIN.R5.Task_ID_Ack=Tracc_TCP AND MAIN.R5.Task_Completed OR GTAC_CONFIG.Option_Robot_Count<5) AND
											(MAIN.R6.Task_ID_Ack=Tracc_TCP AND MAIN.R6.Task_Completed OR GTAC_CONFIG.Option_Robot_Count<6) AND
											(MAIN.R7.Task_ID_Ack=Tracc_TCP AND MAIN.R7.Task_Completed OR GTAC_CONFIG.Option_Robot_Count<7) AND
											(MAIN.R8.Task_ID_Ack=Tracc_TCP AND MAIN.R8.Task_Completed OR GTAC_CONFIG.Option_Robot_Count<8) AND
											(MAIN.R9.Task_ID_Ack=Tracc_TCP AND MAIN.R9.Task_Completed OR GTAC_CONFIG.Option_Robot_Count<9) AND
											(MAIN.R10.Task_ID_Ack=Tracc_TCP AND MAIN.R10.Task_Completed OR GTAC_CONFIG.Option_Robot_Count<10) AND
											(MAIN.R11.Task_ID_Ack=Tracc_TCP AND MAIN.R11.Task_Completed OR GTAC_CONFIG.Option_Robot_Count<11) AND
											(MAIN.R12.Task_ID_Ack=Tracc_TCP AND MAIN.R12.Task_Completed OR GTAC_CONFIG.Option_Robot_Count<12) AND
											(MAIN.R13.Task_ID_Ack=Tracc_TCP AND MAIN.R13.Task_Completed OR GTAC_CONFIG.Option_Robot_Count<13) AND
											(MAIN.R14.Task_ID_Ack=Tracc_TCP AND MAIN.R14.Task_Completed OR GTAC_CONFIG.Option_Robot_Count<14) AND
											(MAIN.R15.Task_ID_Ack=Tracc_TCP AND MAIN.R15.Task_Completed OR GTAC_CONFIG.Option_Robot_Count<15) AND
											(MAIN.R16.Task_ID_Ack=Tracc_TCP AND MAIN.R16.Task_Completed OR GTAC_CONFIG.Option_Robot_Count<16) AND
											(MAIN.R17.Task_ID_Ack=Tracc_TCP AND MAIN.R17.Task_Completed OR GTAC_CONFIG.Option_Robot_Count<17) AND
											(MAIN.R18.Task_ID_Ack=Tracc_TCP AND MAIN.R18.Task_Completed OR GTAC_CONFIG.Option_Robot_Count<18) AND
											(MAIN.R19.Task_ID_Ack=Tracc_TCP AND MAIN.R19.Task_Completed OR GTAC_CONFIG.Option_Robot_Count<19) AND
											(MAIN.R20.Task_ID_Ack=Tracc_TCP AND MAIN.R20.Task_Completed OR GTAC_CONFIG.Option_Robot_Count<20) AND
											(MAIN.R21.Task_ID_Ack=Tracc_TCP AND MAIN.R21.Task_Completed OR GTAC_CONFIG.Option_Robot_Count<21) AND
											(MAIN.R22.Task_ID_Ack=Tracc_TCP AND MAIN.R22.Task_Completed OR GTAC_CONFIG.Option_Robot_Count<22) AND
											(MAIN.R23.Task_ID_Ack=Tracc_TCP AND MAIN.R23.Task_Completed OR GTAC_CONFIG.Option_Robot_Count<23) AND
											(MAIN.R24.Task_ID_Ack=Tracc_TCP AND MAIN.R24.Task_Completed OR GTAC_CONFIG.Option_Robot_Count<24) AND
											(MAIN.R25.Task_ID_Ack=Tracc_TCP AND MAIN.R25.Task_Completed OR GTAC_CONFIG.Option_Robot_Count<25) AND
											(MAIN.R26.Task_ID_Ack=Tracc_TCP AND MAIN.R26.Task_Completed OR GTAC_CONFIG.Option_Robot_Count<26) AND
											(MAIN.R27.Task_ID_Ack=Tracc_TCP AND MAIN.R27.Task_Completed OR GTAC_CONFIG.Option_Robot_Count<27) AND
											(MAIN.R28.Task_ID_Ack=Tracc_TCP AND MAIN.R28.Task_Completed OR GTAC_CONFIG.Option_Robot_Count<28) AND
											(MAIN.R29.Task_ID_Ack=Tracc_TCP AND MAIN.R29.Task_Completed OR GTAC_CONFIG.Option_Robot_Count<29) AND
											(MAIN.R30.Task_ID_Ack=Tracc_TCP AND MAIN.R30.Task_Completed OR GTAC_CONFIG.Option_Robot_Count<30));
											(*ADD MORE*)
	(*Completes for running seperated tip dress jobs*)
	Tip_Dress_Complete1:= MAIN.R1.Task_ID_Ack=Tip_Dress AND MAIN.R1.Task_Completed AND NOT Start_All_TDRobots;
	Tip_Dress_Complete2:= MAIN.R2.Task_ID_Ack=Tip_Dress AND MAIN.R2.Task_Completed AND NOT Start_All_TDRobots;
	Tip_Dress_Complete3:= MAIN.R3.Task_ID_Ack=Tip_Dress AND MAIN.R3.Task_Completed AND NOT Start_All_TDRobots;
	Tip_Dress_Complete4:= MAIN.R4.Task_ID_Ack=Tip_Dress AND MAIN.R4.Task_Completed AND NOT Start_All_TDRobots;
	Tip_Dress_Complete5:= MAIN.R5.Task_ID_Ack=Tip_Dress AND MAIN.R5.Task_Completed AND NOT Start_All_TDRobots;
	Tip_Dress_Complete6:= MAIN.R6.Task_ID_Ack=Tip_Dress AND MAIN.R6.Task_Completed AND NOT Start_All_TDRobots;
	Tip_Dress_Complete7:= MAIN.R7.Task_ID_Ack=Tip_Dress AND MAIN.R7.Task_Completed AND NOT Start_All_TDRobots;
	Tip_Dress_Complete8:= MAIN.R8.Task_ID_Ack=Tip_Dress AND MAIN.R8.Task_Completed AND NOT Start_All_TDRobots;
	Tip_Dress_Complete9:= MAIN.R9.Task_ID_Ack=Tip_Dress AND MAIN.R9.Task_Completed AND NOT Start_All_TDRobots;
	Tip_Dress_Complete10:= MAIN.R10.Task_ID_Ack=Tip_Dress AND MAIN.R10.Task_Completed AND NOT Start_All_TDRobots;
	Tip_Dress_Complete11:= MAIN.R11.Task_ID_Ack=Tip_Dress AND MAIN.R11.Task_Completed AND NOT Start_All_TDRobots;
	Tip_Dress_Complete12:= MAIN.R12.Task_ID_Ack=Tip_Dress AND MAIN.R12.Task_Completed AND NOT Start_All_TDRobots;
	Tip_Dress_Complete13:= MAIN.R13.Task_ID_Ack=Tip_Dress AND MAIN.R13.Task_Completed AND NOT Start_All_TDRobots;
	Tip_Dress_Complete14:= MAIN.R14.Task_ID_Ack=Tip_Dress AND MAIN.R14.Task_Completed AND NOT Start_All_TDRobots;
	Tip_Dress_Complete15:= MAIN.R15.Task_ID_Ack=Tip_Dress AND MAIN.R15.Task_Completed AND NOT Start_All_TDRobots;
	Tip_Dress_Complete16:= MAIN.R16.Task_ID_Ack=Tip_Dress AND MAIN.R16.Task_Completed AND NOT Start_All_TDRobots;
	Tip_Dress_Complete17:= MAIN.R17.Task_ID_Ack=Tip_Dress AND MAIN.R17.Task_Completed AND NOT Start_All_TDRobots;
	Tip_Dress_Complete18:= MAIN.R18.Task_ID_Ack=Tip_Dress AND MAIN.R18.Task_Completed AND NOT Start_All_TDRobots;
	Tip_Dress_Complete19:= MAIN.R19.Task_ID_Ack=Tip_Dress AND MAIN.R19.Task_Completed AND NOT Start_All_TDRobots;
	Tip_Dress_Complete20:= MAIN.R20.Task_ID_Ack=Tip_Dress AND MAIN.R20.Task_Completed AND NOT Start_All_TDRobots;
	Tip_Dress_Complete21:= MAIN.R21.Task_ID_Ack=Tip_Dress AND MAIN.R21.Task_Completed AND NOT Start_All_TDRobots;
	Tip_Dress_Complete22:= MAIN.R22.Task_ID_Ack=Tip_Dress AND MAIN.R22.Task_Completed AND NOT Start_All_TDRobots;
	Tip_Dress_Complete23:= MAIN.R23.Task_ID_Ack=Tip_Dress AND MAIN.R23.Task_Completed AND NOT Start_All_TDRobots;
	Tip_Dress_Complete24:= MAIN.R24.Task_ID_Ack=Tip_Dress AND MAIN.R24.Task_Completed AND NOT Start_All_TDRobots;
	Tip_Dress_Complete25:= MAIN.R25.Task_ID_Ack=Tip_Dress AND MAIN.R25.Task_Completed AND NOT Start_All_TDRobots;
	Tip_Dress_Complete26:= MAIN.R26.Task_ID_Ack=Tip_Dress AND MAIN.R26.Task_Completed AND NOT Start_All_TDRobots;
	Tip_Dress_Complete27:= MAIN.R27.Task_ID_Ack=Tip_Dress AND MAIN.R27.Task_Completed AND NOT Start_All_TDRobots;
	Tip_Dress_Complete28:= MAIN.R28.Task_ID_Ack=Tip_Dress AND MAIN.R28.Task_Completed AND NOT Start_All_TDRobots;
	Tip_Dress_Complete29:= MAIN.R29.Task_ID_Ack=Tip_Dress AND MAIN.R29.Task_Completed AND NOT Start_All_TDRobots;
	Tip_Dress_Complete30:= MAIN.R30.Task_ID_Ack=Tip_Dress AND MAIN.R30.Task_Completed AND NOT Start_All_TDRobots;

	(*Completes for running seperated TraccTCP  jobs*)
	TraccTCP_Complete1:= MAIN.R1.Task_ID_Ack=Tracc_TCP AND MAIN.R1.Task_Completed AND NOT Start_All_TraccTCP;
	TraccTCP_Complete2:= MAIN.R2.Task_ID_Ack=Tracc_TCP AND MAIN.R2.Task_Completed AND NOT Start_All_TraccTCP;
	TraccTCP_Complete3:= MAIN.R3.Task_ID_Ack=Tracc_TCP AND MAIN.R3.Task_Completed AND NOT Start_All_TraccTCP;
	TraccTCP_Complete4:= MAIN.R4.Task_ID_Ack=Tracc_TCP AND MAIN.R4.Task_Completed AND NOT Start_All_TraccTCP;
	TraccTCP_Complete5:= MAIN.R5.Task_ID_Ack=Tracc_TCP AND MAIN.R5.Task_Completed AND NOT Start_All_TraccTCP;
	TraccTCP_Complete6:= MAIN.R6.Task_ID_Ack=Tracc_TCP AND MAIN.R6.Task_Completed AND NOT Start_All_TraccTCP;
	TraccTCP_Complete7:= MAIN.R7.Task_ID_Ack=Tracc_TCP AND MAIN.R7.Task_Completed AND NOT Start_All_TraccTCP;
	TraccTCP_Complete8:= MAIN.R8.Task_ID_Ack=Tracc_TCP AND MAIN.R8.Task_Completed AND NOT Start_All_TraccTCP;
	TraccTCP_Complete9:= MAIN.R9.Task_ID_Ack=Tracc_TCP AND MAIN.R9.Task_Completed AND NOT Start_All_TraccTCP;
	TraccTCP_Complete10:= MAIN.R10.Task_ID_Ack=Tracc_TCP AND MAIN.R10.Task_Completed AND NOT Start_All_TraccTCP;
	TraccTCP_Complete11:= MAIN.R11.Task_ID_Ack=Tracc_TCP AND MAIN.R11.Task_Completed AND NOT Start_All_TraccTCP;
	TraccTCP_Complete12:= MAIN.R12.Task_ID_Ack=Tracc_TCP AND MAIN.R12.Task_Completed AND NOT Start_All_TraccTCP;
	TraccTCP_Complete13:= MAIN.R13.Task_ID_Ack=Tracc_TCP AND MAIN.R13.Task_Completed AND NOT Start_All_TraccTCP;
	TraccTCP_Complete14:= MAIN.R14.Task_ID_Ack=Tracc_TCP AND MAIN.R14.Task_Completed AND NOT Start_All_TraccTCP;
	TraccTCP_Complete15:= MAIN.R15.Task_ID_Ack=Tracc_TCP AND MAIN.R15.Task_Completed AND NOT Start_All_TraccTCP;
	TraccTCP_Complete16:= MAIN.R16.Task_ID_Ack=Tracc_TCP AND MAIN.R16.Task_Completed AND NOT Start_All_TraccTCP;
	TraccTCP_Complete17:= MAIN.R17.Task_ID_Ack=Tracc_TCP AND MAIN.R17.Task_Completed AND NOT Start_All_TraccTCP;
	TraccTCP_Complete18:= MAIN.R18.Task_ID_Ack=Tracc_TCP AND MAIN.R18.Task_Completed AND NOT Start_All_TraccTCP;
	TraccTCP_Complete19:= MAIN.R19.Task_ID_Ack=Tracc_TCP AND MAIN.R19.Task_Completed AND NOT Start_All_TraccTCP;
	TraccTCP_Complete20:= MAIN.R20.Task_ID_Ack=Tracc_TCP AND MAIN.R20.Task_Completed AND NOT Start_All_TraccTCP;
	TraccTCP_Complete21:= MAIN.R21.Task_ID_Ack=Tracc_TCP AND MAIN.R21.Task_Completed AND NOT Start_All_TraccTCP;
	TraccTCP_Complete22:= MAIN.R22.Task_ID_Ack=Tracc_TCP AND MAIN.R22.Task_Completed AND NOT Start_All_TraccTCP;
	TraccTCP_Complete23:= MAIN.R23.Task_ID_Ack=Tracc_TCP AND MAIN.R23.Task_Completed AND NOT Start_All_TraccTCP;
	TraccTCP_Complete24:= MAIN.R24.Task_ID_Ack=Tracc_TCP AND MAIN.R24.Task_Completed AND NOT Start_All_TraccTCP;
	TraccTCP_Complete25:= MAIN.R25.Task_ID_Ack=Tracc_TCP AND MAIN.R25.Task_Completed AND NOT Start_All_TraccTCP;
	TraccTCP_Complete26:= MAIN.R26.Task_ID_Ack=Tracc_TCP AND MAIN.R26.Task_Completed AND NOT Start_All_TraccTCP;
	TraccTCP_Complete27:= MAIN.R27.Task_ID_Ack=Tracc_TCP AND MAIN.R27.Task_Completed AND NOT Start_All_TraccTCP;
	TraccTCP_Complete28:= MAIN.R28.Task_ID_Ack=Tracc_TCP AND MAIN.R28.Task_Completed AND NOT Start_All_TraccTCP;
	TraccTCP_Complete29:= MAIN.R29.Task_ID_Ack=Tracc_TCP AND MAIN.R29.Task_Completed AND NOT Start_All_TraccTCP;
	TraccTCP_Complete30:= MAIN.R30.Task_ID_Ack=Tracc_TCP AND MAIN.R30.Task_Completed AND NOT Start_All_TraccTCP;
	
	(*Data To All Robots*)

	(*Task ID*)
	IF Service_Call_ForAllRobots
		THEN
		R1_Data.Task_ID[16]:=Task_ID;
		R2_Data.Task_ID[16]:=Task_ID;
		R3_Data.Task_ID[16]:=Task_ID;
		R4_Data.Task_ID[16]:=Task_ID;
		R5_Data.Task_ID[16]:=Task_ID;
		R6_Data.Task_ID[16]:=Task_ID;
		R7_Data.Task_ID[16]:=Task_ID;
		R8_Data.Task_ID[16]:=Task_ID;
		R9_Data.Task_ID[16]:=Task_ID;
		R10_Data.Task_ID[16]:=Task_ID;
		R11_Data.Task_ID[16]:=Task_ID;
		R12_Data.Task_ID[16]:=Task_ID;
		R13_Data.Task_ID[16]:=Task_ID;
		R14_Data.Task_ID[16]:=Task_ID;
		R15_Data.Task_ID[16]:=Task_ID;
		R16_Data.Task_ID[16]:=Task_ID;
		R17_Data.Task_ID[16]:=Task_ID;
		R18_Data.Task_ID[16]:=Task_ID;
		R19_Data.Task_ID[16]:=Task_ID;
		R20_Data.Task_ID[16]:=Task_ID;
		R21_Data.Task_ID[16]:=Task_ID;
		R22_Data.Task_ID[16]:=Task_ID;
		R23_Data.Task_ID[16]:=Task_ID;
		R24_Data.Task_ID[16]:=Task_ID;
		R25_Data.Task_ID[16]:=Task_ID;
		R26_Data.Task_ID[16]:=Task_ID;
		R27_Data.Task_ID[16]:=Task_ID;
		R28_Data.Task_ID[16]:=Task_ID;
		R29_Data.Task_ID[16]:=Task_ID;
		R30_Data.Task_ID[16]:=Task_ID;
	END_IF;

	IF Service_Call_ForRobot1 AND Start_TDRobot_1
		THEN
		R1_Data.Task_ID[16]:=Tip_Dress;	
	ELSIF (Service_Call_ForRobot1 AND Start_TraccTCP_1 )
		THEN
		R1_Data.Task_ID[16]:=Tracc_TCP;
	ELSIF NOT Service_Call_ForAllRobots
		THEN
		R1_Data.Task_ID[16]:=0;
	END_IF;

	IF Service_Call_ForRobot2 AND Start_TDRobot_2
		THEN
		R2_Data.Task_ID[16]:=Tip_Dress;
	ELSIF (Service_Call_ForRobot2 AND Start_TraccTCP_2 )
		THEN
		R2_Data.Task_ID[16]:=Tracc_TCP;
	ELSIF NOT Service_Call_ForAllRobots
		THEN
		R2_Data.Task_ID[16]:=0;
	END_IF;

	IF Service_Call_ForRobot3 AND Start_TDRobot_3
		THEN
		R3_Data.Task_ID[16]:=Tip_Dress;
	ELSIF (Service_Call_ForRobot3 AND Start_TraccTCP_3 )
		THEN
		R3_Data.Task_ID[16]:=Tracc_TCP;
	ELSIF NOT Service_Call_ForAllRobots
		THEN
		R3_Data.Task_ID[16]:=0;			
	END_IF;

	IF Service_Call_ForRobot4 AND Start_TDRobot_4
		THEN
		R4_Data.Task_ID[16]:=Tip_Dress;
	ELSIF (Service_Call_ForRobot4 AND Start_TraccTCP_4)
		THEN
		R4_Data.Task_ID[16]:=Tracc_TCP;
	ELSIF NOT Service_Call_ForAllRobots
		THEN
		R4_Data.Task_ID[16]:=0;	
	END_IF;

	IF Service_Call_ForRobot5
		THEN
		R5_Data.Task_ID[16]:=Tip_Dress;
	ELSIF (Service_Call_ForRobot5 AND Start_TraccTCP_5 )
		THEN
		R5_Data.Task_ID[16]:=Tracc_TCP;
	ELSIF NOT Service_Call_ForAllRobots
		THEN
		R5_Data.Task_ID[16]:=0;
	END_IF;

	IF Service_Call_ForRobot6
		THEN
		R6_Data.Task_ID[16]:=Tip_Dress;
	ELSIF (Service_Call_ForRobot6 AND Start_TraccTCP_6 )
		THEN
		R6_Data.Task_ID[16]:=Tracc_TCP;
	ELSIF NOT Service_Call_ForAllRobots
		THEN
		R6_Data.Task_ID[16]:=0;
	END_IF;

	IF Service_Call_ForRobot7
		THEN
		R7_Data.Task_ID[16]:=Tip_Dress;
	ELSIF (Service_Call_ForRobot7 AND Start_TraccTCP_7 )
		THEN
		R7_Data.Task_ID[16]:=Tracc_TCP;
	ELSIF NOT Service_Call_ForAllRobots
		THEN
		R7_Data.Task_ID[16]:=0;
	END_IF;

	IF Service_Call_ForRobot8
		THEN
		R8_Data.Task_ID[16]:=Tip_Dress;
	ELSIF (Service_Call_ForRobot8 AND Start_TraccTCP_8 )
		THEN
		R8_Data.Task_ID[16]:=Tracc_TCP;
	ELSIF NOT Service_Call_ForAllRobots
		THEN
		R8_Data.Task_ID[16]:=0;
	END_IF;

	IF Service_Call_ForRobot9
		THEN
		R9_Data.Task_ID[16]:=Tip_Dress;
	ELSIF (Service_Call_ForRobot9 AND Start_TraccTCP_9 )
		THEN
		R9_Data.Task_ID[16]:=Tracc_TCP;
	ELSIF NOT Service_Call_ForAllRobots
		THEN
		R9_Data.Task_ID[16]:=0;
	END_IF;

	IF Service_Call_ForRobot10
		THEN
		R10_Data.Task_ID[16]:=Tip_Dress;
	ELSIF (Service_Call_ForRobot10 AND Start_TraccTCP_10 )
		THEN
		R10_Data.Task_ID[16]:=Tracc_TCP;
	ELSIF NOT Service_Call_ForAllRobots
		THEN
		R10_Data.Task_ID[16]:=0;
	END_IF;

	IF Service_Call_ForRobot11
		THEN
		R11_Data.Task_ID[16]:=Tip_Dress;
	ELSIF (Service_Call_ForRobot11 AND Start_TraccTCP_11 )
		THEN
		R11_Data.Task_ID[16]:=Tracc_TCP;
	ELSIF NOT Service_Call_ForAllRobots
		THEN
		R11_Data.Task_ID[16]:=0;
	END_IF;

	IF Service_Call_ForRobot12
		THEN
		R12_Data.Task_ID[16]:=Tip_Dress;
	ELSIF (Service_Call_ForRobot12 AND Start_TraccTCP_12 )
		THEN
		R12_Data.Task_ID[16]:=Tracc_TCP;
	ELSIF NOT Service_Call_ForAllRobots
		THEN
		R12_Data.Task_ID[16]:=0;
	END_IF;

	IF Service_Call_ForRobot13
		THEN
		R13_Data.Task_ID[16]:=Tip_Dress;
	ELSIF (Service_Call_ForRobot13 AND Start_TraccTCP_13 )
		THEN
		R13_Data.Task_ID[16]:=Tracc_TCP;
	ELSIF NOT Service_Call_ForAllRobots
		THEN
		R13_Data.Task_ID[16]:=0;
	END_IF;

	IF Service_Call_ForRobot14
		THEN
		R14_Data.Task_ID[16]:=Tip_Dress;
	ELSIF (Service_Call_ForRobot14 AND Start_TraccTCP_14 )
		THEN
		R14_Data.Task_ID[16]:=Tracc_TCP;
	ELSIF NOT Service_Call_ForAllRobots
		THEN
		R14_Data.Task_ID[16]:=0;
	END_IF;

	IF Service_Call_ForRobot15
		THEN
		R15_Data.Task_ID[16]:=Tip_Dress;
	ELSIF (Service_Call_ForRobot15 AND Start_TraccTCP_15 )
		THEN
		R15_Data.Task_ID[16]:=Tracc_TCP;
	ELSIF NOT Service_Call_ForAllRobots
		THEN
		R15_Data.Task_ID[16]:=0;
	END_IF;

	IF Service_Call_ForRobot16
		THEN
		R16_Data.Task_ID[16]:=Tip_Dress;
	ELSIF (Service_Call_ForRobot16 AND Start_TraccTCP_16 )
		THEN
		R16_Data.Task_ID[16]:=Tracc_TCP;
	ELSIF NOT Service_Call_ForAllRobots
		THEN
		R16_Data.Task_ID[16]:=0;
	END_IF;

	IF Service_Call_ForRobot17
		THEN
		R17_Data.Task_ID[16]:=Tip_Dress;
	ELSIF (Service_Call_ForRobot17 AND Start_TraccTCP_17 )
		THEN
		R17_Data.Task_ID[16]:=Tracc_TCP;
	ELSIF NOT Service_Call_ForAllRobots
		THEN
		R17_Data.Task_ID[16]:=0;
	END_IF;

	IF Service_Call_ForRobot18
		THEN
		R18_Data.Task_ID[16]:=Tip_Dress;
	ELSIF (Service_Call_ForRobot18 AND Start_TraccTCP_18 )
		THEN
		R18_Data.Task_ID[16]:=Tracc_TCP;
	ELSIF NOT Service_Call_ForAllRobots
		THEN
		R18_Data.Task_ID[16]:=0;
	END_IF;

	IF Service_Call_ForRobot19
		THEN
		R19_Data.Task_ID[16]:=Tip_Dress;
	ELSIF (Service_Call_ForRobot19 AND Start_TraccTCP_19 )
		THEN
		R19_Data.Task_ID[16]:=Tracc_TCP;
	ELSIF NOT Service_Call_ForAllRobots
		THEN
		R19_Data.Task_ID[16]:=0;
	END_IF;

	IF Service_Call_ForRobot20
		THEN
		R20_Data.Task_ID[16]:=Tip_Dress;
	ELSIF (Service_Call_ForRobot20 AND Start_TraccTCP_20 )
		THEN
		R20_Data.Task_ID[16]:=Tracc_TCP;
	ELSIF NOT Service_Call_ForAllRobots
		THEN
		R20_Data.Task_ID[16]:=0;
	END_IF;

	IF Service_Call_ForRobot21
		THEN
		R21_Data.Task_ID[16]:=Tip_Dress;
	ELSIF (Service_Call_ForRobot21 AND Start_TraccTCP_21 )
		THEN
		R21_Data.Task_ID[16]:=Tracc_TCP;
	ELSIF NOT Service_Call_ForAllRobots
		THEN
		R21_Data.Task_ID[16]:=0;
	END_IF;

	IF Service_Call_ForRobot22
		THEN
		R22_Data.Task_ID[16]:=Tip_Dress;
	ELSIF (Service_Call_ForRobot22 AND Start_TraccTCP_22 )
		THEN
		R22_Data.Task_ID[16]:=Tracc_TCP;
	ELSIF NOT Service_Call_ForAllRobots
		THEN
		R22_Data.Task_ID[16]:=0;
	END_IF;

	IF Service_Call_ForRobot23
		THEN
		R23_Data.Task_ID[16]:=Tip_Dress;
	ELSIF (Service_Call_ForRobot23 AND Start_TraccTCP_23 )
		THEN
		R23_Data.Task_ID[16]:=Tracc_TCP;
	ELSIF NOT Service_Call_ForAllRobots
		THEN
		R23_Data.Task_ID[16]:=0;
	END_IF;

	IF Service_Call_ForRobot24
		THEN
		R24_Data.Task_ID[16]:=Tip_Dress;
	ELSIF (Service_Call_ForRobot24 AND Start_TraccTCP_24 )
		THEN
		R24_Data.Task_ID[16]:=Tracc_TCP;
	ELSIF NOT Service_Call_ForAllRobots
		THEN
		R24_Data.Task_ID[16]:=0;
	END_IF;

	IF Service_Call_ForRobot25
		THEN
		R25_Data.Task_ID[16]:=Tip_Dress;
	ELSIF (Service_Call_ForRobot25 AND Start_TraccTCP_25 )
		THEN
		R25_Data.Task_ID[16]:=Tracc_TCP;
	ELSIF NOT Service_Call_ForAllRobots
		THEN
		R25_Data.Task_ID[16]:=0;
	END_IF;

	IF Service_Call_ForRobot26
		THEN
		R26_Data.Task_ID[16]:=Tip_Dress;
	ELSIF (Service_Call_ForRobot26 AND Start_TraccTCP_26 )
		THEN
		R26_Data.Task_ID[16]:=Tracc_TCP;
	ELSIF NOT Service_Call_ForAllRobots
		THEN
		R26_Data.Task_ID[16]:=0;
	END_IF;

	IF Service_Call_ForRobot27
		THEN
		R27_Data.Task_ID[16]:=Tip_Dress;
	ELSIF (Service_Call_ForRobot27 AND Start_TraccTCP_27 )
		THEN
		R27_Data.Task_ID[16]:=Tracc_TCP;
	ELSIF NOT Service_Call_ForAllRobots
		THEN
		R27_Data.Task_ID[16]:=0;
	END_IF;

	IF Service_Call_ForRobot28
		THEN
		R28_Data.Task_ID[16]:=Tip_Dress;
	ELSIF (Service_Call_ForRobot28 AND Start_TraccTCP_28 )
		THEN
		R28_Data.Task_ID[16]:=Tracc_TCP;
	ELSIF NOT Service_Call_ForAllRobots
		THEN
		R28_Data.Task_ID[16]:=0;
	END_IF;

	IF Service_Call_ForRobot29
		THEN
		R29_Data.Task_ID[16]:=Tip_Dress;
	ELSIF (Service_Call_ForRobot29 AND Start_TraccTCP_29 )
		THEN
		R29_Data.Task_ID[16]:=Tracc_TCP;
	ELSIF NOT Service_Call_ForAllRobots
		THEN
		R29_Data.Task_ID[16]:=0;
	END_IF;

	IF Service_Call_ForRobot30
		THEN
		R30_Data.Task_ID[16]:=Tip_Dress;
	ELSIF (Service_Call_ForRobot30 AND Start_TraccTCP_30 )
		THEN
		R30_Data.Task_ID[16]:=Tracc_TCP;
	ELSIF NOT Service_Call_ForAllRobots
		THEN
		R30_Data.Task_ID[16]:=0;
	END_IF;

	(*Fix ID*)
	R1_Data.Fix_ID[16]:= Fix_ID;
	R2_Data.Fix_ID[16]:= Fix_ID;
	R3_Data.Fix_ID[16]:= Fix_ID;
	R4_Data.Fix_ID[16]:= Fix_ID;
	R5_Data.Fix_ID[16]:= Fix_ID;
	R6_Data.Fix_ID[16]:= Fix_ID;
	R7_Data.Fix_ID[16]:= Fix_ID;
	R8_Data.Fix_ID[16]:= Fix_ID;
	R9_Data.Fix_ID[16]:= Fix_ID;
	R10_Data.Fix_ID[16]:= Fix_ID;
	R11_Data.Fix_ID[16]:= Fix_ID;
	R12_Data.Fix_ID[16]:= Fix_ID;
	R13_Data.Fix_ID[16]:= Fix_ID;
	R14_Data.Fix_ID[16]:= Fix_ID;
	R15_Data.Fix_ID[16]:= Fix_ID;
	R16_Data.Fix_ID[16]:= Fix_ID;
	R17_Data.Fix_ID[16]:= Fix_ID;
	R18_Data.Fix_ID[16]:= Fix_ID;
	R19_Data.Fix_ID[16]:= Fix_ID;
	R20_Data.Fix_ID[16]:= Fix_ID;
	R21_Data.Fix_ID[16]:= Fix_ID;
	R22_Data.Fix_ID[16]:= Fix_ID;
	R23_Data.Fix_ID[16]:= Fix_ID;
	R24_Data.Fix_ID[16]:= Fix_ID;
	R25_Data.Fix_ID[16]:= Fix_ID;
	R26_Data.Fix_ID[16]:= Fix_ID;
	R27_Data.Fix_ID[16]:= Fix_ID;
	R28_Data.Fix_ID[16]:= Fix_ID;
	R29_Data.Fix_ID[16]:= Fix_ID;
	R30_Data.Fix_ID[16]:= Fix_ID;

	(*Model ID*)
	R1_Data.Model_ID[16]:= Model_ID;
	R2_Data.Model_ID[16]:= Model_ID;
	R3_Data.Model_ID[16]:= Model_ID;
	R4_Data.Model_ID[16]:= Model_ID;
	R5_Data.Model_ID[16]:= Model_ID;
	R6_Data.Model_ID[16]:= Model_ID;
	R7_Data.Model_ID[16]:= Model_ID;
	R8_Data.Model_ID[16]:= Model_ID;
	R9_Data.Model_ID[16]:= Model_ID;
	R10_Data.Model_ID[16]:= Model_ID;
	R11_Data.Model_ID[16]:= Model_ID;
	R12_Data.Model_ID[16]:= Model_ID;
	R13_Data.Model_ID[16]:= Model_ID;
	R14_Data.Model_ID[16]:= Model_ID;
	R15_Data.Model_ID[16]:= Model_ID;
	R16_Data.Model_ID[16]:= Model_ID;
	R17_Data.Model_ID[16]:= Model_ID;
	R18_Data.Model_ID[16]:= Model_ID;
	R19_Data.Model_ID[16]:= Model_ID;
	R20_Data.Model_ID[16]:= Model_ID;
	R21_Data.Model_ID[16]:= Model_ID;
	R22_Data.Model_ID[16]:= Model_ID;
	R23_Data.Model_ID[16]:= Model_ID;
	R24_Data.Model_ID[16]:= Model_ID;
	R25_Data.Model_ID[16]:= Model_ID;
	R26_Data.Model_ID[16]:= Model_ID;
	R27_Data.Model_ID[16]:= Model_ID;
	R28_Data.Model_ID[16]:= Model_ID;
	R29_Data.Model_ID[16]:= Model_ID;
	R30_Data.Model_ID[16]:= Model_ID;

	(*Proceed from Pounce*)
	R1_Data.Proceed_From_Pounce[16]:= Robots_Clear_ToProceed OR (Service_Call_ForRobot1);
	R2_Data.Proceed_From_Pounce[16]:= Robots_Clear_ToProceed OR (Service_Call_ForRobot2);
	R3_Data.Proceed_From_Pounce[16]:= Robots_Clear_ToProceed OR (Service_Call_ForRobot3);
	R4_Data.Proceed_From_Pounce[16]:= Robots_Clear_ToProceed OR (Service_Call_ForRobot4);
	R5_Data.Proceed_From_Pounce[16]:= Robots_Clear_ToProceed OR (Service_Call_ForRobot5);
	R6_Data.Proceed_From_Pounce[16]:= Robots_Clear_ToProceed OR (Service_Call_ForRobot6);
	R7_Data.Proceed_From_Pounce[16]:= Robots_Clear_ToProceed OR (Service_Call_ForRobot7);
	R8_Data.Proceed_From_Pounce[16]:= Robots_Clear_ToProceed OR (Service_Call_ForRobot8);
	R9_Data.Proceed_From_Pounce[16]:= Robots_Clear_ToProceed OR (Service_Call_ForRobot9);
	R10_Data.Proceed_From_Pounce[16]:= Robots_Clear_ToProceed OR (Service_Call_ForRobot10);
	R11_Data.Proceed_From_Pounce[16]:= Robots_Clear_ToProceed OR (Service_Call_ForRobot11);
	R12_Data.Proceed_From_Pounce[16]:= Robots_Clear_ToProceed OR (Service_Call_ForRobot12);
	R13_Data.Proceed_From_Pounce[16]:= Robots_Clear_ToProceed OR (Service_Call_ForRobot13);
	R14_Data.Proceed_From_Pounce[16]:= Robots_Clear_ToProceed OR (Service_Call_ForRobot14);
	R15_Data.Proceed_From_Pounce[16]:= Robots_Clear_ToProceed OR (Service_Call_ForRobot15);
	R16_Data.Proceed_From_Pounce[16]:= Robots_Clear_ToProceed OR (Service_Call_ForRobot16);
	R17_Data.Proceed_From_Pounce[16]:= Robots_Clear_ToProceed OR (Service_Call_ForRobot17);
	R18_Data.Proceed_From_Pounce[16]:= Robots_Clear_ToProceed OR (Service_Call_ForRobot18);
	R19_Data.Proceed_From_Pounce[16]:= Robots_Clear_ToProceed OR (Service_Call_ForRobot19);
	R20_Data.Proceed_From_Pounce[16]:= Robots_Clear_ToProceed OR (Service_Call_ForRobot20);
	R21_Data.Proceed_From_Pounce[16]:= Robots_Clear_ToProceed OR (Service_Call_ForRobot21);
	R22_Data.Proceed_From_Pounce[16]:= Robots_Clear_ToProceed OR (Service_Call_ForRobot22);
	R23_Data.Proceed_From_Pounce[16]:= Robots_Clear_ToProceed OR (Service_Call_ForRobot23);
	R24_Data.Proceed_From_Pounce[16]:= Robots_Clear_ToProceed OR (Service_Call_ForRobot24);
	R25_Data.Proceed_From_Pounce[16]:= Robots_Clear_ToProceed OR (Service_Call_ForRobot25);
	R26_Data.Proceed_From_Pounce[16]:= Robots_Clear_ToProceed OR (Service_Call_ForRobot26);
	R27_Data.Proceed_From_Pounce[16]:= Robots_Clear_ToProceed OR (Service_Call_ForRobot27);
	R28_Data.Proceed_From_Pounce[16]:= Robots_Clear_ToProceed OR (Service_Call_ForRobot28);
	R29_Data.Proceed_From_Pounce[16]:= Robots_Clear_ToProceed OR (Service_Call_ForRobot29);
	R30_Data.Proceed_From_Pounce[16]:= Robots_Clear_ToProceed OR (Service_Call_ForRobot30);

	(*Complete Acks*)
	R1_Data.Complete_Ack[16]:=All_Complete_Ack OR (Tip_Dress_Complete1) OR TraccTCP_Complete1;
	R2_Data.Complete_Ack[16]:=All_Complete_Ack OR (Tip_Dress_Complete2) OR TraccTCP_Complete2;
	R3_Data.Complete_Ack[16]:=All_Complete_Ack OR (Tip_Dress_Complete3) OR TraccTCP_Complete3;
	R4_Data.Complete_Ack[16]:=All_Complete_Ack OR (Tip_Dress_Complete4) OR TraccTCP_Complete4;
	R5_Data.Complete_Ack[16]:=All_Complete_Ack OR (Tip_Dress_Complete5) OR TraccTCP_Complete5;
	R6_Data.Complete_Ack[16]:=All_Complete_Ack OR (Tip_Dress_Complete6) OR TraccTCP_Complete6;
	R7_Data.Complete_Ack[16]:=All_Complete_Ack OR (Tip_Dress_Complete7) OR TraccTCP_Complete7;
	R8_Data.Complete_Ack[16]:=All_Complete_Ack OR (Tip_Dress_Complete8) OR TraccTCP_Complete8;
	R9_Data.Complete_Ack[16]:=All_Complete_Ack OR (Tip_Dress_Complete9) OR TraccTCP_Complete9;
	R10_Data.Complete_Ack[16]:=All_Complete_Ack OR (Tip_Dress_Complete10) OR TraccTCP_Complete10;
	R11_Data.Complete_Ack[16]:=All_Complete_Ack OR (Tip_Dress_Complete11) OR TraccTCP_Complete11;
	R12_Data.Complete_Ack[16]:=All_Complete_Ack OR (Tip_Dress_Complete12) OR TraccTCP_Complete12;
	R13_Data.Complete_Ack[16]:=All_Complete_Ack OR (Tip_Dress_Complete13) OR TraccTCP_Complete13;
	R14_Data.Complete_Ack[16]:=All_Complete_Ack OR (Tip_Dress_Complete14) OR TraccTCP_Complete14;
	R15_Data.Complete_Ack[16]:=All_Complete_Ack OR (Tip_Dress_Complete15) OR TraccTCP_Complete15;
	R16_Data.Complete_Ack[16]:=All_Complete_Ack OR (Tip_Dress_Complete16) OR TraccTCP_Complete16;
	R17_Data.Complete_Ack[16]:=All_Complete_Ack OR (Tip_Dress_Complete17) OR TraccTCP_Complete17;
	R18_Data.Complete_Ack[16]:=All_Complete_Ack OR (Tip_Dress_Complete18) OR TraccTCP_Complete18;
	R19_Data.Complete_Ack[16]:=All_Complete_Ack OR (Tip_Dress_Complete19) OR TraccTCP_Complete19;
	R20_Data.Complete_Ack[16]:=All_Complete_Ack OR (Tip_Dress_Complete20) OR TraccTCP_Complete20;
	R21_Data.Complete_Ack[16]:=All_Complete_Ack OR (Tip_Dress_Complete21) OR TraccTCP_Complete21;
	R22_Data.Complete_Ack[16]:=All_Complete_Ack OR (Tip_Dress_Complete22) OR TraccTCP_Complete22;
	R23_Data.Complete_Ack[16]:=All_Complete_Ack OR (Tip_Dress_Complete23) OR TraccTCP_Complete23;
	R24_Data.Complete_Ack[16]:=All_Complete_Ack OR (Tip_Dress_Complete24) OR TraccTCP_Complete24;
	R25_Data.Complete_Ack[16]:=All_Complete_Ack OR (Tip_Dress_Complete25) OR TraccTCP_Complete25;
	R26_Data.Complete_Ack[16]:=All_Complete_Ack OR (Tip_Dress_Complete26) OR TraccTCP_Complete26;
	R27_Data.Complete_Ack[16]:=All_Complete_Ack OR (Tip_Dress_Complete27) OR TraccTCP_Complete27;
	R28_Data.Complete_Ack[16]:=All_Complete_Ack OR (Tip_Dress_Complete28) OR TraccTCP_Complete28;
	R29_Data.Complete_Ack[16]:=All_Complete_Ack OR (Tip_Dress_Complete29) OR TraccTCP_Complete29;
	R30_Data.Complete_Ack[16]:=All_Complete_Ack OR (Tip_Dress_Complete30) OR TraccTCP_Complete30;

	(*Peripheral Req Acks*)
	R1_Data.PeripheralReq_Ack[16]:= Repo_Ack;
	
	IF MAIN.R1.Task_ID_Ack=Tip_Dress THEN
		R1_Data.PeripheralReq_Ack[16].1 := MAIN.R1.Peripheral_Req.1 AND MAIN.R1.Reamer[1].Ream_Delay.Q  AND MAIN.R1.Reamer[1].Ream_Clamp_Open; 
		R1_Data.PeripheralReq_Ack[16].2 := MAIN.R1.Peripheral_Req.2 AND MAIN.R1.Reamer[1].Spray_Delay.Q; 
		R1_Data.PeripheralReq_Ack[16].4 := MAIN.R1.Peripheral_Req.4 AND MAIN.R1.Reamer[1].WireCutter_Delay.Q; 
	END_IF
	
	R2_Data.PeripheralReq_Ack[16]:= Repo_Ack;
	
	IF MAIN.R2.Task_ID_Ack=Tip_Dress THEN
		R2_Data.PeripheralReq_Ack[16].1 := MAIN.R2.Peripheral_Req.1 AND MAIN.R2.Reamer[1].Ream_Delay.Q AND MAIN.R2.Reamer[1].Ream_Clamp_Open; 
		R2_Data.PeripheralReq_Ack[16].2 := MAIN.R2.Peripheral_Req.2 AND MAIN.R2.Reamer[1].Spray_Delay.Q; 
		R2_Data.PeripheralReq_Ack[16].4 := MAIN.R2.Peripheral_Req.4 AND MAIN.R2.Reamer[1].WireCutter_Delay.Q; 
	END_IF
	
	R3_Data.PeripheralReq_Ack[16]:= Repo_Ack;
	
	IF MAIN.R3.Task_ID_Ack=Tip_Dress THEN
		R3_Data.PeripheralReq_Ack[16].1 := MAIN.R3.Peripheral_Req.1 AND MAIN.R3.Reamer[1].Ream_Delay.Q AND MAIN.R3.Reamer[1].Ream_Clamp_Open; 
		R3_Data.PeripheralReq_Ack[16].2 := MAIN.R3.Peripheral_Req.2 AND MAIN.R3.Reamer[1].Spray_Delay.Q; 
		R3_Data.PeripheralReq_Ack[16].4 := MAIN.R3.Peripheral_Req.4 AND MAIN.R3.Reamer[1].WireCutter_Delay.Q; 
	END_IF
	
	R5_Data.PeripheralReq_Ack[16]:= Repo_Ack;
	
	IF MAIN.R5.Task_ID_Ack=Tip_Dress THEN
		R5_Data.PeripheralReq_Ack[16].1 := MAIN.R5.Peripheral_Req.1 AND MAIN.R5.Reamer[1].Ream_Delay.Q AND MAIN.R5.Reamer[1].Ream_Clamp_Open; 
		R5_Data.PeripheralReq_Ack[16].2 := MAIN.R5.Peripheral_Req.2 AND MAIN.R5.Reamer[1].Spray_Delay.Q; 
		R5_Data.PeripheralReq_Ack[16].4 := MAIN.R5.Peripheral_Req.4 AND MAIN.R5.Reamer[1].WireCutter_Delay.Q; 
	END_IF
	
	R6_Data.PeripheralReq_Ack[16]:= Repo_Ack;
	
	IF MAIN.R6.Task_ID_Ack=Tip_Dress THEN
		R6_Data.PeripheralReq_Ack[16].1 := MAIN.R6.Peripheral_Req.1 AND MAIN.R6.Reamer[1].Ream_Delay.Q AND MAIN.R6.Reamer[1].Ream_Clamp_Open; 
		R6_Data.PeripheralReq_Ack[16].2 := MAIN.R6.Peripheral_Req.2 AND MAIN.R6.Reamer[1].Spray_Delay.Q; 
		R6_Data.PeripheralReq_Ack[16].4 := MAIN.R6.Peripheral_Req.4 AND MAIN.R6.Reamer[1].WireCutter_Delay.Q; 
	END_IF
	
	R7_Data.PeripheralReq_Ack[16]:= Repo_Ack;
	
	IF MAIN.R7.Task_ID_Ack=Tip_Dress THEN
		R7_Data.PeripheralReq_Ack[16].1 := MAIN.R7.Peripheral_Req.1 AND MAIN.R7.Reamer[1].Ream_Delay.Q AND MAIN.R7.Reamer[1].Ream_Clamp_Open; 
		R7_Data.PeripheralReq_Ack[16].2 := MAIN.R7.Peripheral_Req.2 AND MAIN.R7.Reamer[1].Spray_Delay.Q; 
		R7_Data.PeripheralReq_Ack[16].4 := MAIN.R7.Peripheral_Req.4 AND MAIN.R7.Reamer[1].WireCutter_Delay.Q; 
	END_IF
	
	R8_Data.PeripheralReq_Ack[16]:= Repo_Ack;
	
	IF MAIN.R8.Task_ID_Ack=Tip_Dress THEN
		R8_Data.PeripheralReq_Ack[16].1 := MAIN.R8.Peripheral_Req.1 AND MAIN.R8.Reamer[1].Ream_Delay.Q AND MAIN.R8.Reamer[1].Ream_Clamp_Open; 
		R8_Data.PeripheralReq_Ack[16].2 := MAIN.R8.Peripheral_Req.2 AND MAIN.R8.Reamer[1].Spray_Delay.Q; 
		R8_Data.PeripheralReq_Ack[16].4 := MAIN.R8.Peripheral_Req.4 AND MAIN.R8.Reamer[1].WireCutter_Delay.Q; 
	END_IF
	
	R9_Data.PeripheralReq_Ack[16]:= Repo_Ack;
	
	IF MAIN.R9.Task_ID_Ack=Tip_Dress THEN
		R9_Data.PeripheralReq_Ack[16].1 := MAIN.R9.Peripheral_Req.1 AND MAIN.R9.Reamer[1].Ream_Delay.Q AND MAIN.R9.Reamer[1].Ream_Clamp_Open; 
		R9_Data.PeripheralReq_Ack[16].2 := MAIN.R9.Peripheral_Req.2 AND MAIN.R9.Reamer[1].Spray_Delay.Q; 
		R9_Data.PeripheralReq_Ack[16].4 := MAIN.R9.Peripheral_Req.4 AND MAIN.R9.Reamer[1].WireCutter_Delay.Q; 
	END_IF
	

	R4_Data.PeripheralReq_Ack[16]:= Repo_Ack;
	R10_Data.PeripheralReq_Ack[16]:= Repo_Ack;
	R11_Data.PeripheralReq_Ack[16]:= Repo_Ack;
	R12_Data.PeripheralReq_Ack[16]:= Repo_Ack;
	R13_Data.PeripheralReq_Ack[16]:= Repo_Ack;
	R14_Data.PeripheralReq_Ack[16]:= Repo_Ack;
	R15_Data.PeripheralReq_Ack[16]:= Repo_Ack;
	R16_Data.PeripheralReq_Ack[16]:= Repo_Ack;
	R17_Data.PeripheralReq_Ack[16]:= Repo_Ack;
	R18_Data.PeripheralReq_Ack[16]:= Repo_Ack;
	R19_Data.PeripheralReq_Ack[16]:= Repo_Ack;
	R20_Data.PeripheralReq_Ack[16]:= Repo_Ack;
	R21_Data.PeripheralReq_Ack[16]:= Repo_Ack;
	R22_Data.PeripheralReq_Ack[16]:= Repo_Ack;
	R23_Data.PeripheralReq_Ack[16]:= Repo_Ack;
	R24_Data.PeripheralReq_Ack[16]:= Repo_Ack;
	R25_Data.PeripheralReq_Ack[16]:= Repo_Ack;
	R26_Data.PeripheralReq_Ack[16]:= Repo_Ack;
	R27_Data.PeripheralReq_Ack[16]:= Repo_Ack;
	R28_Data.PeripheralReq_Ack[16]:= Repo_Ack;
	R29_Data.PeripheralReq_Ack[16]:= Repo_Ack;
	R30_Data.PeripheralReq_Ack[16]:= Repo_Ack;

(*%%%%%%%%%%%%%% Call Robots to Tool and Give Them, Task ID, Fixture ID and Model ID %%%%%%%%%%%%%%%%%*)

	(* Perform Call To Service*)
	Service_Call_ForAllRobots:= (Start_All_MTRobots AND NOT Start_All_BTRobots AND NOT Start_All_TCRobots)
								OR (NOT Start_All_MTRobots AND Start_All_BTRobots AND NOT Start_All_TCRobots)
								OR (NOT Start_All_MTRobots AND NOT Start_All_BTRobots AND Start_All_TCRobots);

	Service_Call_ForRobot1:= (Start_TDRobot_1 OR Start_TraccTCP_1) AND NOT Start_All_MTRobots AND NOT Start_All_BTRobots AND NOT Start_All_TCRobots;
	Service_Call_ForRobot2:= (Start_TDRobot_2 OR Start_TraccTCP_2) AND NOT Start_All_MTRobots AND NOT Start_All_BTRobots AND NOT Start_All_TCRobots;
	Service_Call_ForRobot3:= (Start_TDRobot_3 OR Start_TraccTCP_3) AND NOT Start_All_MTRobots AND NOT Start_All_BTRobots AND NOT Start_All_TCRobots;
	Service_Call_ForRobot4:= (Start_TDRobot_4 OR Start_TraccTCP_4) AND NOT Start_All_MTRobots AND NOT Start_All_BTRobots AND NOT Start_All_TCRobots;
	Service_Call_ForRobot5:= (Start_TDRobot_5 OR Start_TraccTCP_5) AND NOT Start_All_MTRobots AND NOT Start_All_BTRobots AND NOT Start_All_TCRobots;
	Service_Call_ForRobot6:= (Start_TDRobot_6 OR Start_TraccTCP_6) AND NOT Start_All_MTRobots AND NOT Start_All_BTRobots AND NOT Start_All_TCRobots;
	Service_Call_ForRobot7:= (Start_TDRobot_7 OR Start_TraccTCP_7) AND NOT Start_All_MTRobots AND NOT Start_All_BTRobots AND NOT Start_All_TCRobots;
	Service_Call_ForRobot8:= (Start_TDRobot_8 OR Start_TraccTCP_8) AND NOT Start_All_MTRobots AND NOT Start_All_BTRobots AND NOT Start_All_TCRobots;
	Service_Call_ForRobot9:= (Start_TDRobot_9 OR Start_TraccTCP_9) AND NOT Start_All_MTRobots AND NOT Start_All_BTRobots AND NOT Start_All_TCRobots;
	Service_Call_ForRobot10:= (Start_TDRobot_10 OR Start_TraccTCP_10) AND NOT Start_All_MTRobots AND NOT Start_All_BTRobots AND NOT Start_All_TCRobots;
	Service_Call_ForRobot11:= (Start_TDRobot_11 OR Start_TraccTCP_11) AND NOT Start_All_MTRobots AND NOT Start_All_BTRobots AND NOT Start_All_TCRobots;
	Service_Call_ForRobot12:= (Start_TDRobot_12 OR Start_TraccTCP_12) AND NOT Start_All_MTRobots AND NOT Start_All_BTRobots AND NOT Start_All_TCRobots;
	Service_Call_ForRobot13:= (Start_TDRobot_13 OR Start_TraccTCP_13) AND NOT Start_All_MTRobots AND NOT Start_All_BTRobots AND NOT Start_All_TCRobots;
	Service_Call_ForRobot14:= (Start_TDRobot_14 OR Start_TraccTCP_14) AND NOT Start_All_MTRobots AND NOT Start_All_BTRobots AND NOT Start_All_TCRobots;
	Service_Call_ForRobot15:= (Start_TDRobot_15 OR Start_TraccTCP_15) AND NOT Start_All_MTRobots AND NOT Start_All_BTRobots AND NOT Start_All_TCRobots;
	Service_Call_ForRobot16:= (Start_TDRobot_16 OR Start_TraccTCP_16) AND NOT Start_All_MTRobots AND NOT Start_All_BTRobots AND NOT Start_All_TCRobots;
	Service_Call_ForRobot17:= (Start_TDRobot_17 OR Start_TraccTCP_17) AND NOT Start_All_MTRobots AND NOT Start_All_BTRobots AND NOT Start_All_TCRobots;
	Service_Call_ForRobot18:= (Start_TDRobot_18 OR Start_TraccTCP_18) AND NOT Start_All_MTRobots AND NOT Start_All_BTRobots AND NOT Start_All_TCRobots;
	Service_Call_ForRobot19:= (Start_TDRobot_19 OR Start_TraccTCP_19) AND NOT Start_All_MTRobots AND NOT Start_All_BTRobots AND NOT Start_All_TCRobots;
	Service_Call_ForRobot20:= (Start_TDRobot_20 OR Start_TraccTCP_20) AND NOT Start_All_MTRobots AND NOT Start_All_BTRobots AND NOT Start_All_TCRobots;
	Service_Call_ForRobot21:= (Start_TDRobot_21 OR Start_TraccTCP_21) AND NOT Start_All_MTRobots AND NOT Start_All_BTRobots AND NOT Start_All_TCRobots;
	Service_Call_ForRobot22:= (Start_TDRobot_22 OR Start_TraccTCP_22) AND NOT Start_All_MTRobots AND NOT Start_All_BTRobots AND NOT Start_All_TCRobots;
	Service_Call_ForRobot23:= (Start_TDRobot_23 OR Start_TraccTCP_23) AND NOT Start_All_MTRobots AND NOT Start_All_BTRobots AND NOT Start_All_TCRobots;
	Service_Call_ForRobot24:= (Start_TDRobot_24 OR Start_TraccTCP_24) AND NOT Start_All_MTRobots AND NOT Start_All_BTRobots AND NOT Start_All_TCRobots;
	Service_Call_ForRobot25:= (Start_TDRobot_25 OR Start_TraccTCP_25) AND NOT Start_All_MTRobots AND NOT Start_All_BTRobots AND NOT Start_All_TCRobots;
	Service_Call_ForRobot26:= (Start_TDRobot_26 OR Start_TraccTCP_26) AND NOT Start_All_MTRobots AND NOT Start_All_BTRobots AND NOT Start_All_TCRobots;
	Service_Call_ForRobot27:= (Start_TDRobot_27 OR Start_TraccTCP_27) AND NOT Start_All_MTRobots AND NOT Start_All_BTRobots AND NOT Start_All_TCRobots;
	Service_Call_ForRobot28:= (Start_TDRobot_28 OR Start_TraccTCP_28) AND NOT Start_All_MTRobots AND NOT Start_All_BTRobots AND NOT Start_All_TCRobots;
	Service_Call_ForRobot29:= (Start_TDRobot_29 OR Start_TraccTCP_29) AND NOT Start_All_MTRobots AND NOT Start_All_BTRobots AND NOT Start_All_TCRobots;
	Service_Call_ForRobot30:= (Start_TDRobot_30 OR Start_TraccTCP_30) AND NOT Start_All_MTRobots AND NOT Start_All_BTRobots AND NOT Start_All_TCRobots;

	(*Allow Robots to Proceed Into Tool*)
	(*!!!!!This is the final OK to allow Robots Into the Tool Area, So it Better Be Ready!!!!!!!*)
	IF Enable_Motion
		THEN
			IF (All_MTRobots_Proceed OR All_BTRobots_Proceed OR All_TCRobots_Proceed OR All_TraccTCP_Proceed) AND All_Robots_WorkingOK
				THEN Robots_Clear_ToProceed:=TRUE;
				ELSE Robots_Clear_ToProceed:= FALSE;
			END_IF;
		ELSE Robots_Clear_ToProceed:= FALSE;
	END_IF;

	(*Develop Task IDs - See Global Variable, "TaskID_Record"*)

	IF Start_All_MTRobots AND Enable_Motion
		THEN
			Task_ID:= Master_Test;
	ELSIF Start_All_BTRobots AND Enable_Motion
		THEN
			Task_ID:= Brake_Test;
	ELSIF Start_All_TCRobots AND Enable_Motion
		THEN
			Task_ID:= Tip_Change;
	ELSIF Start_All_TDRobots AND Enable_Motion
		THEN
			Task_ID:= Tip_Dress;
	ELSIF Start_TDRobot_1 AND Enable_Motion
		THEN
			Task_ID:= Tip_Dress;
	ELSIF Start_TDRobot_2 AND Enable_Motion
		THEN
			Task_ID:= Tip_Dress;
	ELSIF Start_TDRobot_3 AND Enable_Motion
		THEN
			Task_ID:= Tip_Dress;
	ELSIF Start_TDRobot_4 AND Enable_Motion
		THEN
			Task_ID:= Tip_Dress;
	ELSIF Start_TDRobot_5 AND Enable_Motion
		THEN
			Task_ID:= Tip_Dress;
	ELSIF Start_TDRobot_6 AND Enable_Motion
		THEN
			Task_ID:= Tip_Dress;
	ELSIF Start_TDRobot_7 AND Enable_Motion
		THEN
			Task_ID:= Tip_Dress;
	ELSIF Start_TDRobot_8 AND Enable_Motion
		THEN
			Task_ID:= Tip_Dress;
	ELSIF Start_TDRobot_9 AND Enable_Motion
		THEN
			Task_ID:= Tip_Dress;
	ELSIF Start_TDRobot_10 AND Enable_Motion
		THEN
			Task_ID:= Tip_Dress;
	ELSIF Start_TDRobot_11 AND Enable_Motion
		THEN
			Task_ID:= Tip_Dress;
	ELSIF Start_TDRobot_12 AND Enable_Motion
		THEN
			Task_ID:= Tip_Dress;
	ELSIF Start_TDRobot_13 AND Enable_Motion
		THEN
			Task_ID:= Tip_Dress;
	ELSIF Start_TDRobot_14 AND Enable_Motion
		THEN
			Task_ID:= Tip_Dress;
	ELSIF Start_TDRobot_15 AND Enable_Motion
		THEN
			Task_ID:= Tip_Dress;
	ELSIF Start_TDRobot_16 AND Enable_Motion
		THEN
			Task_ID:= Tip_Dress;
	ELSIF Start_TDRobot_17 AND Enable_Motion
		THEN
			Task_ID:= Tip_Dress;
	ELSIF Start_TDRobot_18 AND Enable_Motion
		THEN
			Task_ID:= Tip_Dress;
	ELSIF Start_TDRobot_19 AND Enable_Motion
		THEN
			Task_ID:= Tip_Dress;
	ELSIF Start_TDRobot_20 AND Enable_Motion
		THEN
			Task_ID:= Tip_Dress;
	ELSIF Start_TDRobot_21 AND Enable_Motion
		THEN
			Task_ID:= Tip_Dress;
	ELSIF Start_TDRobot_22 AND Enable_Motion
		THEN
			Task_ID:= Tip_Dress;
	ELSIF Start_TDRobot_23 AND Enable_Motion
		THEN
			Task_ID:= Tip_Dress;
	ELSIF Start_TDRobot_24 AND Enable_Motion
		THEN
			Task_ID:= Tip_Dress;
	ELSIF Start_TDRobot_25 AND Enable_Motion
		THEN
			Task_ID:= Tip_Dress;
	ELSIF Start_TDRobot_26 AND Enable_Motion
		THEN
			Task_ID:= Tip_Dress;
	ELSIF Start_TDRobot_27 AND Enable_Motion
		THEN
			Task_ID:= Tip_Dress;
	ELSIF Start_TDRobot_28 AND Enable_Motion
		THEN
			Task_ID:= Tip_Dress;
	ELSIF Start_TDRobot_29 AND Enable_Motion
		THEN
			Task_ID:= Tip_Dress;
	ELSIF Start_TDRobot_30 AND Enable_Motion
		THEN
			Task_ID:= Tip_Dress;
	ELSIF Start_TraccTCP_1 AND Enable_Motion
		THEN
			Task_ID:= Tracc_TCP;
	ELSIF Start_TraccTCP_2 AND Enable_Motion
		THEN
			Task_ID:= Tracc_TCP;
	ELSIF Start_TraccTCP_3 AND Enable_Motion
		THEN
			Task_ID:= Tracc_TCP;
	ELSIF Start_TraccTCP_4 AND Enable_Motion
		THEN
			Task_ID:= Tracc_TCP;		
(*ADD MORE*)			
	ELSE Task_ID:= 0;
	END_IF;



	(*Develop Fixture ID*)
	Fix_ID:= 1;					(*In Future Map Beckhoff Dip Switch Data From IP67 Block to Here*)
	(*Develop Model ID*)
	Model_ID:= Discrete_In.ModelData;		(*1 = AB Ring 4DR, 2 = AB Ring 5DR*)


(*+++++++++++++++++++++++++++++++++++++++++++++++ Task Complete Acks ++++++++++++++++++++++++++*)

	(*Complete Ack*)
	All_Complete_Ack:= All_Robots_Complete AND Cycle_Complete;



(*!!!!!!!!!!!!!!!!!!!!!!!!!!!!!!!!!!!!!!!!!!!!!!!!!!!!!!!!!!!!!!!!!!!!!!!!!!!!!!!!!!!!!!!! Tool Repositions !!!!!!!!!!!!!!!!!!!!!!!!!!!!!!!!!!!!!!!!!!!!!!!!!!!!!!!!!!!!!!!!!!!!!!!!!!!!!!!!!!!!!!!!!!!*)
(*+++++++++++THIS AREA IS CUSTOM PER INSTALLATION AND WILL HAVE TO BE MODIFIED PER +++++++++++++*)
(*+++++++++++THIS AREA IS CUSTOM PER INSTALLATION AND WILL HAVE TO BE MODIFIED PER +++++++++++++*)

	(*Reposition Request#1*)
	IF MAIN.R1.Task_ID_Ack=Tip_Change AND MAIN.R1.Peripheral_Req.0 AND
		(MAIN.R2.Task_ID_Ack=Tip_Change AND MAIN.R2.Peripheral_Req.0 OR GTAC_CONFIG.Option_Robot_Count<2) AND
		(MAIN.R3.Task_ID_Ack=Tip_Change AND MAIN.R3.Peripheral_Req.0 OR GTAC_CONFIG.Option_Robot_Count<3) AND
		(MAIN.R4.Task_ID_Ack=Tip_Change AND MAIN.R4.Peripheral_Req.0 OR GTAC_CONFIG.Option_Robot_Count<4) AND
		(MAIN.R5.Task_ID_Ack=Tip_Change AND MAIN.R5.Peripheral_Req.0 OR GTAC_CONFIG.Option_Robot_Count<5) AND
		(MAIN.R6.Task_ID_Ack=Tip_Change AND MAIN.R6.Peripheral_Req.0 OR GTAC_CONFIG.Option_Robot_Count<6) AND
		(MAIN.R7.Task_ID_Ack=Tip_Change AND MAIN.R7.Peripheral_Req.0 OR GTAC_CONFIG.Option_Robot_Count<7) AND
		(MAIN.R8.Task_ID_Ack=Tip_Change AND MAIN.R8.Peripheral_Req.0 OR GTAC_CONFIG.Option_Robot_Count<8) AND
		(MAIN.R9.Task_ID_Ack=Tip_Change AND MAIN.R9.Peripheral_Req.0 OR GTAC_CONFIG.Option_Robot_Count<9) AND
		(MAIN.R10.Task_ID_Ack=Tip_Change AND MAIN.R10.Peripheral_Req.0 OR GTAC_CONFIG.Option_Robot_Count<10) AND
		(MAIN.R11.Task_ID_Ack=Tip_Change AND MAIN.R11.Peripheral_Req.0 OR GTAC_CONFIG.Option_Robot_Count<11) AND
		(MAIN.R12.Task_ID_Ack=Tip_Change AND MAIN.R12.Peripheral_Req.0 OR GTAC_CONFIG.Option_Robot_Count<12) AND
		(MAIN.R13.Task_ID_Ack=Tip_Change AND MAIN.R13.Peripheral_Req.0 OR GTAC_CONFIG.Option_Robot_Count<13) AND
		(MAIN.R14.Task_ID_Ack=Tip_Change AND MAIN.R14.Peripheral_Req.0 OR GTAC_CONFIG.Option_Robot_Count<14) AND
		(MAIN.R15.Task_ID_Ack=Tip_Change AND MAIN.R15.Peripheral_Req.0 OR GTAC_CONFIG.Option_Robot_Count<15) AND
		(MAIN.R16.Task_ID_Ack=Tip_Change AND MAIN.R16.Peripheral_Req.0 OR GTAC_CONFIG.Option_Robot_Count<16) AND
		(MAIN.R17.Task_ID_Ack=Tip_Change AND MAIN.R17.Peripheral_Req.0 OR GTAC_CONFIG.Option_Robot_Count<17) AND
		(MAIN.R18.Task_ID_Ack=Tip_Change AND MAIN.R18.Peripheral_Req.0 OR GTAC_CONFIG.Option_Robot_Count<18) AND
		(MAIN.R19.Task_ID_Ack=Tip_Change AND MAIN.R19.Peripheral_Req.0 OR GTAC_CONFIG.Option_Robot_Count<19) AND
		(MAIN.R20.Task_ID_Ack=Tip_Change AND MAIN.R20.Peripheral_Req.0 OR GTAC_CONFIG.Option_Robot_Count<20) AND
		(MAIN.R21.Task_ID_Ack=Tip_Change AND MAIN.R21.Peripheral_Req.0 OR GTAC_CONFIG.Option_Robot_Count<21) AND
		(MAIN.R22.Task_ID_Ack=Tip_Change AND MAIN.R22.Peripheral_Req.0 OR GTAC_CONFIG.Option_Robot_Count<22) AND
		(MAIN.R23.Task_ID_Ack=Tip_Change AND MAIN.R23.Peripheral_Req.0 OR GTAC_CONFIG.Option_Robot_Count<23) AND
		(MAIN.R24.Task_ID_Ack=Tip_Change AND MAIN.R24.Peripheral_Req.0 OR GTAC_CONFIG.Option_Robot_Count<24) AND
		(MAIN.R25.Task_ID_Ack=Tip_Change AND MAIN.R25.Peripheral_Req.0 OR GTAC_CONFIG.Option_Robot_Count<25) AND
		(MAIN.R26.Task_ID_Ack=Tip_Change AND MAIN.R26.Peripheral_Req.0 OR GTAC_CONFIG.Option_Robot_Count<26) AND
		(MAIN.R27.Task_ID_Ack=Tip_Change AND MAIN.R27.Peripheral_Req.0 OR GTAC_CONFIG.Option_Robot_Count<27) AND
		(MAIN.R28.Task_ID_Ack=Tip_Change AND MAIN.R28.Peripheral_Req.0 OR GTAC_CONFIG.Option_Robot_Count<28) AND
		(MAIN.R29.Task_ID_Ack=Tip_Change AND MAIN.R29.Peripheral_Req.0 OR GTAC_CONFIG.Option_Robot_Count<29) AND
		(MAIN.R30.Task_ID_Ack=Tip_Change AND MAIN.R30.Peripheral_Req.0 OR GTAC_CONFIG.Option_Robot_Count<30)
		THEN
			Repo_Reqs.0:= TRUE;
	END_IF;
	(*Reposition Request#2*)
	IF (MAIN.R1.Peripheral_Req.1) AND (MAIN.R1.Task_ID_Ack=Tip_Dress)
		THEN
			Repo_Reqs.1:= TRUE;
	END_IF;
	(*Reposition Request#3*)
	IF (MAIN.R2.Peripheral_Req.2) AND (MAIN.R2.Task_ID_Ack=Tip_Dress)
		THEN
			Repo_Reqs.2:= TRUE;
	END_IF;
	(*Reposition Request#4*)
	IF (MAIN.R3.Peripheral_Req.3) AND (MAIN.R3.Task_ID_Ack=Tip_Dress)
		THEN
			Repo_Reqs.3:= TRUE;
	END_IF;
	(*Reposition Request#5*)
	IF (MAIN.R4.Peripheral_Req.4) AND (MAIN.R4.Task_ID_Ack=Tip_Dress)
		THEN
			Repo_Reqs.4:= TRUE;
	END_IF;
	(*----Add more as required-----*)
	(*----Add more as required-----*)


	(*Reset All Reposition Acks At the End Of Cycle*)
	IF Cycle_Complete
		THEN
			Repo_Reqs:= 0;
	END_IF;
(*------------------------- Reposition Acks ---------------------*)
	Repo_Ack.0:= Repo_Reqs.0 AND In_From_ICxx.TipChange_Complete;
	(*Debug - Example of reamer. adjust to the robot as needed. this is setup for a fronius reamer
	Repo_Ack.1:= Repo_Reqs.1 AND MAIN.R2.Reamer[1].WireCutter_ACK AND (MAIN.R2.Task_ID_Ack=Tip_Dress); 
	Repo_Ack.2:= Repo_Reqs.2 AND MAIN.R2.Reamer[1].Injector_ACK AND (MAIN.R2.Task_ID_Ack=Tip_Dress);
	Repo_Ack.3:= Repo_Reqs.3 AND MAIN.R2.Reamer[1].LifterUp_ACK AND (MAIN.R2.Task_ID_Ack=Tip_Dress);
	Repo_Ack.4:= Repo_Reqs.4 AND MAIN.R2.Reamer[1].Clamp_ACK AND (MAIN.R2.Task_ID_Ack=Tip_Dress);
	Repo_ACk.5:= Repo_Reqs.5 AND MAIN.R2.Reamer[1].Reaming_Complete AND (MAIN.R2.Task_ID_Ack=Tip_Dress);*)

(*------------------------ Reposition Visualization --------------------------*)
	Rxx_ReadyAt_TipChangePosition.1:= MAIN.R1.Task_ID_Ack=Tip_Change AND MAIN.R1.Peripheral_Req.0;
	Rxx_ReadyAt_TipChangePosition.2:= MAIN.R2.Task_ID_Ack=Tip_Change AND MAIN.R2.Peripheral_Req.0;
	Rxx_ReadyAt_TipChangePosition.3:= MAIN.R3.Task_ID_Ack=Tip_Change AND MAIN.R3.Peripheral_Req.0;
	Rxx_ReadyAt_TipChangePosition.4:= MAIN.R4.Task_ID_Ack=Tip_Change AND MAIN.R4.Peripheral_Req.0;
	Rxx_ReadyAt_TipChangePosition.5:= MAIN.R5.Task_ID_Ack=Tip_Change AND MAIN.R5.Peripheral_Req.0;
	Rxx_ReadyAt_TipChangePosition.6:= MAIN.R6.Task_ID_Ack=Tip_Change AND MAIN.R6.Peripheral_Req.0;
	Rxx_ReadyAt_TipChangePosition.7:= MAIN.R7.Task_ID_Ack=Tip_Change AND MAIN.R7.Peripheral_Req.0;
	Rxx_ReadyAt_TipChangePosition.8:= MAIN.R8.Task_ID_Ack=Tip_Change AND MAIN.R8.Peripheral_Req.0;
	Rxx_ReadyAt_TipChangePosition.9:= MAIN.R9.Task_ID_Ack=Tip_Change AND MAIN.R9.Peripheral_Req.0;
	Rxx_ReadyAt_TipChangePosition.10:= MAIN.R10.Task_ID_Ack=Tip_Change AND MAIN.R10.Peripheral_Req.0;
	Rxx_ReadyAt_TipChangePosition.11:= MAIN.R11.Task_ID_Ack=Tip_Change AND MAIN.R11.Peripheral_Req.0;
	Rxx_ReadyAt_TipChangePosition.12:= MAIN.R12.Task_ID_Ack=Tip_Change AND MAIN.R12.Peripheral_Req.0;
	Rxx_ReadyAt_TipChangePosition.13:= MAIN.R13.Task_ID_Ack=Tip_Change AND MAIN.R13.Peripheral_Req.0;
	Rxx_ReadyAt_TipChangePosition.14:= MAIN.R14.Task_ID_Ack=Tip_Change AND MAIN.R14.Peripheral_Req.0;
	Rxx_ReadyAt_TipChangePosition.15:= MAIN.R15.Task_ID_Ack=Tip_Change AND MAIN.R15.Peripheral_Req.0;
	Rxx_ReadyAt_TipChangePosition.16:= MAIN.R16.Task_ID_Ack=Tip_Change AND MAIN.R16.Peripheral_Req.0;
	Rxx_ReadyAt_TipChangePosition.17:= MAIN.R17.Task_ID_Ack=Tip_Change AND MAIN.R17.Peripheral_Req.0;
	Rxx_ReadyAt_TipChangePosition.18:= MAIN.R18.Task_ID_Ack=Tip_Change AND MAIN.R18.Peripheral_Req.0;
	Rxx_ReadyAt_TipChangePosition.19:= MAIN.R19.Task_ID_Ack=Tip_Change AND MAIN.R19.Peripheral_Req.0;
	Rxx_ReadyAt_TipChangePosition.20:= MAIN.R20.Task_ID_Ack=Tip_Change AND MAIN.R20.Peripheral_Req.0;
	Rxx_ReadyAt_TipChangePosition.21:= MAIN.R21.Task_ID_Ack=Tip_Change AND MAIN.R21.Peripheral_Req.0;
	Rxx_ReadyAt_TipChangePosition.22:= MAIN.R22.Task_ID_Ack=Tip_Change AND MAIN.R22.Peripheral_Req.0;
	Rxx_ReadyAt_TipChangePosition.23:= MAIN.R23.Task_ID_Ack=Tip_Change AND MAIN.R23.Peripheral_Req.0;
	Rxx_ReadyAt_TipChangePosition.24:= MAIN.R24.Task_ID_Ack=Tip_Change AND MAIN.R24.Peripheral_Req.0;
	Rxx_ReadyAt_TipChangePosition.25:= MAIN.R25.Task_ID_Ack=Tip_Change AND MAIN.R25.Peripheral_Req.0;
	Rxx_ReadyAt_TipChangePosition.26:= MAIN.R26.Task_ID_Ack=Tip_Change AND MAIN.R26.Peripheral_Req.0;
	Rxx_ReadyAt_TipChangePosition.27:= MAIN.R27.Task_ID_Ack=Tip_Change AND MAIN.R27.Peripheral_Req.0;
	Rxx_ReadyAt_TipChangePosition.28:= MAIN.R28.Task_ID_Ack=Tip_Change AND MAIN.R28.Peripheral_Req.0;
	Rxx_ReadyAt_TipChangePosition.29:= MAIN.R29.Task_ID_Ack=Tip_Change AND MAIN.R29.Peripheral_Req.0;
	Rxx_ReadyAt_TipChangePosition.30:= MAIN.R30.Task_ID_Ack=Tip_Change AND MAIN.R30.Peripheral_Req.0;
	Rxx_ReadyAt_TipChangePosition.0:= Repo_Reqs.0;

(*?????????????????????????????????????????????????????????????????????????????????????????????????????????????????????????????????*)

(*$$$$$$$$$$$$$$$$$$$$$$$$$$$$$$$$$$$$$$$$$$$$$$$$$$$ Faults $$$$$$$$$$$$$$$$$$$$$$$$$$$$$$$$$$$$$$$$$$$$$$$$$$$$$$$*)

(*$$$$$$$$$$$$$$$$$$$$$$$$$$$$$$$$$$$$$$$$$$$$$$ Transfer Standard Outputs $$$$$$$$$$$$$$$$$$$$$$$$$$$$$$$$$$$$$$$$$$$*)

(*$$$$$$$$$$$$$$$$$$$$$$$$$$$$$$$$$$$$$$$$$$$$$$ Transfer Safety Outputs $$$$$$$$$$$$$$$$$$$$$$$$$$$$$$$$$$$$$$$$$$$*)

END_PROGRAM

// ---- POUs/Misc/Task_ID_Record.TcPOU
(*
	Revisions
	************
	November 2014
		- added TaskID for sweeping fixtures if they are turn tables
*)

PROGRAM Task_ID_Record
VAR_INPUT
	Enable_Prog: BOOL;

END_VAR

VAR

END_VAR

VAR_OUTPUT
	Prog_Ok: BOOL;
END_VAR

Prog_OK:= TRUE;

(*--------------------------------------------------------------------------------------- Set Static Variables for Comparative Use In Program ------------------------------------------*)
		(*All Task IDs*)
		Dropoff_Fix01:=10;
		Weld_Fix01:=11;						(*Changed to allow different types of robots to work with existing code*)
		Pickup_Fix01:=12;
		Seal_Fix01:=13;
		Stud_Fix01:=14;
		Sweep_Fix01 := 15;

		Dropoff_Fix02:=20;
		Weld_Fix02:=21;							(*Changed to allow different types of robots to work with existing code*)
		Pickup_Fix02:=22;
		Seal_Fix02:=23;
		Stud_Fix02:=24;
		Sweep_Fix02 := 25;

		Dropoff_Fix03:=30;
		Weld_Fix03:=31;
		Pickup_Fix03:=32;
		Seal_Fix03:=33;
		Stud_Fix03:=34;
		Sweep_Fix03 := 35;

		Dropoff_FiX04:=40;
		Weld_Fix04:=41;
		Pickup_Fix04:=42;
		Seal_Fix04:=43;
		Stud_Fix04:=44;
		Sweep_Fix04 := 45;

		Dropoff_Fix05:=50;
		Weld_Fix05:=51;
		Pickup_Fix05:=52;
		Seal_Fix05:=53;
		Stud_Fix05:=54;
		Sweep_Fix05 := 55;

		Dropoff_Fix06:=60;
		Weld_Fix06:=61;
		Pickup_Fix06:=62;
		Seal_Fix06:=63;
		Stud_Fix06:=64;
		Sweep_Fix06 := 65;

		Dropoff_Fix07:=70;
		Weld_Fix07:=71;
		Pickup_Fix07:=72;
		Seal_Fix07:=73;
		Stud_Fix07:=74;
		Sweep_Fix07 := 75;

